Yaskawa INFORM job: X2_57-69(1)(90,0)_HARDOX.JBI

/JOB
//NAME X2_57-69(1)(90,0)_HARDOX
//POS
///NPOS 575,575,575,36,0,0
///TOOL 0
///POSTYPE PULSE
///PULSE
C00000=1941,-102693,-129564,10,101994,-18
C00001=-114160,-110711,-132276,13468,99543,32658
C00002=-115352,64839,21503,33302,71092,28193
C00003=-108531,78392,43986,16123,55140,37786
C00004=-108866,85252,55178,17040,51979,37122
C00005=-108996,88365,60166,17472,50599,36819
C00006=-108995,88536,62039,17737,49581,36632
C00007=-109034,88718,61766,17697,49840,36662
C00008=-109565,92254,66229,18307,49070,36272
C00009=-109034,88718,61766,17697,49840,36662
C00010=-108904,85509,56654,17244,51243,36976
C00011=-108571,78466,45235,16289,54445,37659
C00012=-107997,64928,29160,15382,57165,38310
C00013=-122208,49017,56535,29995,44799,-20500
C00014=-121054,58896,69591,30976,41821,-21001
C00015=-120607,61403,73283,31313,40811,-21157
C00016=-120607,63170,76793,32085,39739,-21613
C00017=-120607,62274,75028,31694,40274,-21383
C00018=-120608,64965,78215,32056,39778,-21596
C00019=-120607,62274,75028,31694,40274,-21383
C00020=-121364,56707,67057,30894,42308,-20982
C00021=-122534,47142,54464,30007,45185,-20534
C00022=-121995,48000,54847,25969,42983,-17450
C00023=-121016,58047,68030,26856,40021,-17900
C00024=-120639,62684,74202,27406,38635,-18182
C00025=-120639,64991,78769,28376,37190,-18734
C00026=-120639,62684,74202,27406,38635,-18182
C00027=-120856,61874,74409,27857,38220,-18464
C00028=-120445,66454,79858,28202,37199,-18614
C00029=-120856,61874,74409,27857,38220,-18464
C00030=-121238,57224,68232,27288,39602,-18174
C00031=-122229,47153,55046,26369,42553,-17714
C00032=-125892,1211,1187,22441,56600,-15676
C00033=-137814,-110158,-69296,24031,60757,-19595
C00034=-137728,-112604,-73316,23755,61850,-19313
C00035=-105364,-57557,-72999,2137,103390,46474
C00036=-115634,-1069,-31686,2185,107255,43060
C00037=-118085,-9413,-35378,2154,105305,42191
C00038=-118085,-9697,-34142,2144,104400,42176
C00039=-118085,-9660,-34317,2144,104526,42177
C00040=-119256,-9729,-34371,2141,104555,41779
C00041=-118897,-9712,-34357,2142,104546,41900
C00042=-118842,-14639,-38555,2142,104596,41919
C00043=-120602,-14747,-38323,2136,104444,41320
C00044=-120602,-13691,-37523,2136,104492,41320
C00045=-120602,-14272,-38765,2141,104957,41329
C00046=-118914,16972,-18491,2200,108489,41969
C00047=-117885,44382,12736,2123,103335,42227
C00048=-118751,44086,13966,2114,102449,41917
C00049=-118751,43916,15366,2106,101498,41903
C00050=-118751,43947,15080,2107,101690,41906
C00051=-119535,43897,15027,2105,101717,41640
C00052=-118660,44084,14052,2114,102390,41948
C00053=-117266,9455,-21352,2173,106346,42489
C00054=-117960,10005,-18871,2157,105121,42232
C00055=-117960,9788,-17905,2150,104416,42222
C00056=-117960,9832,-18111,2152,104564,42225
C00057=-119133,9750,-18184,2151,104599,41827
C00058=-118065,10242,-19838,2168,105841,42211
C00059=-118344,37722,-10535,2304,114239,18149
C00060=-118344,37722,-10535,2304,114239,-9791
C00061=-118344,37722,-10535,2304,91932,-69227
C00062=-118057,36728,-9901,-15898,90565,-72906
C00063=-124690,36878,-9748,-13863,89447,-74870
C00064=-125711,47870,427,-20022,100421,-78286
C00065=-126617,46625,2928,-19712,98166,-78212
C00066=-126617,46154,3748,-19667,97464,-78100
C00067=-126616,46214,3639,-19671,97560,-78116
C00068=-126105,44250,1538,-19774,97945,-78006
C00069=-130834,16270,-22947,-10503,81163,-76491
C00070=-130240,16776,-22499,-10733,81221,-76303
C00071=-130834,16571,-23478,-10493,81637,-76531
C00072=-131370,9383,-27977,-16260,78843,-76537
C00073=-131370,8975,-27154,-16296,78153,-76446
C00074=-131370,9027,-27263,-16291,78243,-76458
C00075=-131518,11566,-25004,-16235,78132,-76492
C00076=-131370,9027,-27263,-16291,78243,-76458
C00077=-132977,7860,-28293,-15633,77980,-76959
C00078=-131370,9307,-27828,-16266,78716,-76522
C00079=-122012,12842,-31502,-19803,84485,-74326
C00080=-122012,12842,-31502,-19803,84485,-74326
C00081=-119946,1839,-34459,-20715,81343,-73118
C00082=-119946,1422,-33631,-20749,80663,-73001
C00083=-119946,1471,-33732,-20744,80745,-73014
C00084=-120414,3746,-31827,-20569,80632,-73154
C00085=-119946,1471,-33731,-20744,80745,-73014
C00086=-130666,4901,-34214,-1657,83498,-73725
C00087=-129717,5880,-33367,-2009,83503,-73430
C00088=-120411,3435,-35647,-20479,82691,-73505
C00089=-123377,35712,-8759,-20752,103203,-78015
C00090=-123377,35712,-8759,-20752,103203,-78015
C00091=-123377,35151,-7898,-20672,102434,-77880
C00092=-123377,35217,-8004,-20682,102528,-77896
C00093=-123032,33253,-10001,-20749,102814,-77829
C00094=-123377,35217,-8004,-20682,102528,-77896
C00095=-124617,7277,-31513,-18537,87356,-75496
C00096=-125486,6411,-32266,-18262,87197,-75758
C00097=-124034,25111,-19103,-19892,98282,-77292
C00098=-138286,19736,-25230,-18597,101765,-82781
C00099=-139019,19392,-24177,-18406,100832,-82879
C00100=-139019,19048,-23693,-18372,100380,-82810
C00101=-139019,19115,-23789,-18378,100469,-82824
C00102=-138733,16890,-25865,-18440,100655,-82756
C00103=-139019,19115,-23789,-18378,100469,-82824
C00104=-148681,-9689,-46202,-1769,83169,-81630
C00105=-147538,-9148,-45777,-2193,83212,-81274
C00106=-148681,-9489,-46523,-1768,83469,-81634
C00107=-146164,-19217,-50920,-12366,76791,-81583
C00108=-146164,-19609,-50092,-12399,76095,-81512
C00109=-146164,-19552,-50218,-12394,76199,-81523
C00110=-146291,-17352,-48598,-12332,76313,-81579
C00111=-146227,-19942,-50503,-12369,76166,-81540
C00112=-147006,-20177,-50674,-12036,76040,-81783
C00113=-147897,-20398,-50837,-11655,75903,-82065
C00114=-147006,-19883,-51298,-12011,76564,-81835
C00115=-146427,-15690,-53542,-12122,80105,-82001
C00116=-146969,1425,-40243,-1367,79119,-79945
C00117=-144686,1127,-36373,-2406,76633,-79189
C00118=-144686,503,-35222,-2413,75606,-79175
C00119=-144686,641,-35492,-2413,75844,-79178
C00120=-144296,-3511,-38926,-2590,75836,-79052
C00121=-144296,-3690,-38579,-2592,75529,-79045
C00122=-144498,-2214,-37368,-2500,75537,-79111
C00123=-144701,-2831,-40035,-2396,76857,-79201
C00124=-153238,-15902,-45841,-12806,65800,-84378
C00125=-152617,-17217,-44336,-13318,64330,-83987
C00126=-152617,-17517,-43346,-13402,63584,-83898
C00127=-152617,-17437,-43619,-13378,63789,-83922
C00128=-152421,-22078,-47006,-13522,63527,-83819
C00129=-152421,-22202,-46551,-13563,63190,-83778
C00130=-152438,-20565,-45369,-13541,63298,-83797
C00131=-152580,-20987,-46826,-13385,63937,-83926
C00132=-154783,-40455,-61981,-12201,62944,-84616
C00133=-154783,-40864,-60420,-12327,61798,-84491
C00134=-154783,-41124,-59200,-12428,60934,-84393
C00135=-154783,-41063,-59504,-12403,61147,-84418
C00136=-152360,-40978,-59451,-13805,61537,-83550
C00137=-152360,-41066,-58995,-13847,61219,-83509
C00138=-153473,-40883,-58880,-13201,61064,-83911
C00139=-153098,-40967,-60326,-13315,61948,-83876
C00140=-169234,-16286,-61298,12968,85350,-87708
C00141=-176944,51771,6509,16270,80043,-90766
C00142=-175584,58970,15892,12405,82098,-90729
C00143=-175584,58471,16898,12427,81244,-90815
C00144=-175584,58538,16756,12423,81362,-90803
C00145=-175497,61195,19784,12406,80863,-90825
C00146=-175583,58538,16759,12438,81362,-90802
C00147=-168381,55909,13794,-5779,79883,-75223
C00148=-169176,56215,14138,-5481,79777,-75473
C00149=-168381,56447,12778,-5766,80781,-75265
C00150=-168717,73846,30007,3804,89205,-89178
C00151=-168717,73499,30710,3804,88596,-89198
C00152=-168717,73540,30620,3804,88675,-89193
C00153=-168793,71056,27634,3823,89235,-89202
C00154=-168717,73540,30620,3804,88675,-89193
C00155=-173050,67061,24969,13193,85810,-87576
C00156=-172324,66679,24524,12986,85777,-87344
C00157=-173050,67500,24071,13186,86568,-87495
C00158=-159020,60616,9002,-2431,101880,-86822
C00159=-158791,58641,10338,-2451,100051,-86715
C00160=-158791,57927,11282,-2444,99105,-86700
C00161=-158791,58001,11179,-2444,99208,-86703
C00162=-158877,55601,8473,-2433,99638,-86739
C00163=-158791,58001,11179,-2444,99208,-86703
C00164=-166389,29268,-13939,12099,84481,-87034
C00165=-165362,29139,-14065,11731,84356,-86720
C00166=-166389,29843,-14777,12087,85274,-86957
C00167=-168101,32508,-13251,8701,86943,-88153
C00168=-168101,31796,-12263,8703,85980,-88221
C00169=-168101,31909,-12426,8703,86137,-88210
C00170=-168113,34589,-9708,8710,85845,-88235
C00171=-167998,32289,-12043,8668,86088,-88180
C00172=-162647,21052,-20406,-2140,79162,-88550
C00173=-163390,21250,-20220,-1826,79131,-88783
C00174=-162647,21510,-21118,-2136,79834,-88562
C00175=-171713,88888,42294,-4924,102711,-49051
C00176=-183434,69304,21781,-4068,104650,-52979
C00177=-184172,69401,22560,-3999,104187,-53203
C00178=-184172,68923,23286,-3988,103496,-53177
C00179=-184172,68963,23221,-3991,103557,-53179
C00180=-183398,68489,22559,-4056,103756,-52932
C00181=-184172,68963,23221,-3991,103557,-53179
C00182=-173144,55424,11916,-25339,98078,-53030
C00183=-173306,53739,10045,-25337,98292,-53134
C00184=-184172,68963,23221,-3991,103557,-53179
C00185=-174683,52284,7590,-20558,90834,-51552
C00186=-174683,51681,8611,-20548,89951,-51401
C00187=-174683,51761,8468,-20549,90073,-51423
C00188=-175494,52416,9191,-20335,89781,-51643
C00189=-174683,51761,8468,-20549,90073,-51423
C00190=-174543,53466,10356,-20583,89839,-51336
C00191=-174438,56042,13238,-20604,89444,-51233
C00192=-174543,54156,9188,-20598,90847,-51507
C00193=-160426,19849,-34491,-24758,102852,-49155
C00194=-102402,-48698,-67991,2144,104784,47502
C00195=-177118,-86899,-49314,70294,69346,55717
C00196=-162665,-62437,-38431,68363,61957,60420
C00197=-158949,-60049,-34374,68890,58994,60353
C00198=-157479,-59004,-32692,69121,57826,60324
C00199=-157483,-57954,-30366,69642,57492,59876
C00200=-157504,-58291,-30998,69516,57587,59981
C00201=-155795,-59629,-31689,69630,56353,60099
C00202=-157504,-58291,-30998,69516,57587,59981
C00203=-157484,-58197,-30924,69514,57575,59985
C00204=-156523,-55844,-29677,69224,57103,60350
C00205=-157484,-58197,-30924,69514,57575,59985
C00206=-162670,-61686,-36716,68690,61698,60098
C00207=-161856,-67053,-41033,60813,38521,63477
C00208=-158996,-62210,-35558,60803,36300,63693
C00209=-157898,-60236,-33315,60834,35435,63760
C00210=-157901,-59173,-30986,61942,34994,63152
C00211=-156769,-58533,-30874,61190,34419,63655
C00212=-156166,-58108,-30651,60848,34087,63889
C00213=-156769,-58791,-31436,60917,34526,63803
C00214=-161883,-66170,-39058,61667,38156,62985
C00215=-175307,-91794,-54277,68294,45083,57713
C00216=-192656,-55134,-37587,64210,60039,59083
C00217=-162159,-23717,-10104,69718,77823,43469
C00218=-159534,-21701,-5637,70155,75421,43047
C00219=-158490,-20805,-3772,70360,74468,42873
C00220=-158493,-19842,-1317,70611,74104,42419
C00221=-158430,-19960,-1760,70561,74138,42521
C00222=-157077,-18912,-994,70615,73251,42719
C00223=-158430,-19960,-1760,70561,74138,42521
C00224=-162097,-22978,-8198,69866,77487,43129
C00225=-164656,-6441,2331,68796,80646,40119
C00226=-162354,-4355,7073,69146,78392,39620
C00227=-161441,-2725,10948,69469,77194,39063
C00228=-161443,-1987,12871,69626,76894,38710
C00229=-161439,-2551,11387,69503,77124,38984
C00230=-160415,-1923,12464,69637,76311,38965
C00231=-159548,-1589,12743,69678,75730,39076
C00232=-160719,-2768,10769,69490,76742,39193
C00233=-164702,-5497,5223,68969,80178,39553
C00234=-192656,-55134,-37587,64210,60039,59083
C00235=-125486,-104854,-75041,22917,86800,-65584
C00236=-126033,-92220,-87194,23391,99857,-63257
C00237=-126008,-87407,-69757,22927,92227,-64737
C00238=-122771,-89042,-67284,23124,89141,-64144
C00239=-121425,-89554,-66224,23215,87919,-63888
C00240=-121418,-87602,-63818,23218,87477,-63971
C00241=-121371,-87768,-64101,23220,87545,-63941
C00242=-119041,-87737,-64090,23370,86898,-63214
C00243=-121371,-87768,-64101,23220,87545,-63941
C00244=-119842,-88584,-64995,23320,87236,-63441
C00245=-119807,-91269,-65466,23334,86221,-63626
C00246=-119842,-88584,-64995,23320,87236,-63441
C00247=-121199,-88128,-66077,23230,88448,-63702
C00248=-124465,-86636,-68609,23034,91510,-64308
C00249=-142854,-85767,-72329,35934,81198,-48667
C00250=-140267,-86079,-63689,45810,58760,-32657
C00251=-135996,-80956,-60126,44498,56909,-31284
C00252=-134384,-78850,-58646,43955,56229,-30750
C00253=-134256,-77036,-56222,44175,55757,-30924
C00254=-134288,-77408,-56713,44133,55854,-30891
C00255=-132164,-77894,-56932,43544,54718,-30303
C00256=-134288,-77408,-56713,44133,55854,-30891
C00257=-88320,-91033,-56979,-46001,31828,15275
C00258=-89280,-88900,-56774,-44237,32046,14267
C00259=-88320,-91033,-56979,-46001,31828,15275
C00260=-85210,-101515,-62011,-50678,31900,18023
C00261=-89666,-105996,-71374,-46997,57370,39665
C00262=-112926,-92756,-65130,-39557,61499,44934
C00263=-117841,-88867,-61535,-38560,59130,43528
C00264=-119732,-87223,-60045,-38129,58240,42969
C00265=-119742,-85223,-57591,-38309,57852,43124
C00266=-119765,-85676,-58172,-38256,57941,43076
C00267=-121812,-86923,-58375,-37936,56635,42605
C00268=-119765,-85676,-58172,-38256,57941,43076
C00269=-121275,-85554,-58782,-37706,57631,42461
C00270=-122404,-83336,-58379,-37071,57860,41818
C00271=-121275,-85554,-58782,-37706,57631,42461
C00272=-114616,-91226,-63955,-39185,60786,44412
C00273=-114645,-97965,-79407,-37345,65578,42515
C00274=-116729,-83918,-76551,-18553,86191,61698
C00275=-117159,-89242,-76095,-11181,89587,70256
C00276=-119083,-90759,-73003,-11190,86687,69852
C00277=-119889,-89726,-70248,-11201,85432,69686
C00278=-119897,-88175,-68603,-11203,85218,69702
C00279=-119889,-89726,-70248,-11201,85432,69686
C00280=-119873,-91603,-70614,-11208,84708,69757
C00281=-119889,-89726,-70248,-11201,85432,69686
C00282=-107060,-93796,-69139,-19617,83326,67746
C00283=-109561,-94345,-69347,-19648,82582,66969
C00284=-107060,-93796,-69139,-19617,83326,67746
C00285=-120981,-91693,-72872,-11196,85873,69270
C00286=-118990,-90334,-76042,-11186,88750,69699
C00287=-119015,-93571,-89875,-11280,95471,69085
C00288=-121827,-98987,-110994,4235,90756,33976
C00289=-126467,-111869,-98615,30475,51467,-26148
C00290=-122938,-103029,-94111,27808,51796,-24337
C00291=-121643,-99583,-92275,26825,51945,-23680
C00292=-121634,-97826,-90039,26985,51518,-23798
C00293=-121643,-99583,-92275,26825,51945,-23680
C00294=-130783,-80407,-84869,35916,67887,-27578
C00295=-128717,-80853,-85070,35145,66956,-27002
C00296=-130783,-80407,-84869,35916,67887,-27578
C00297=-107674,-109601,-92730,7088,37825,-14001
C00298=-108083,-105924,-92018,7248,39302,-14088
C00299=-107674,-109601,-92730,7088,37825,-14001
C00300=-110011,-124661,-99237,10171,34381,-15732
C00301=-126906,-107253,-113226,22382,79753,-37979
C00302=-126893,-93432,-102362,29867,101882,-55415
C00303=-122864,-96655,-100816,29402,98217,-54829
C00304=-121215,-97700,-100096,29236,96792,-54563
C00305=-121210,-96197,-97952,29195,96310,-54685
C00306=-121215,-97700,-100096,29236,96792,-54563
C00307=-121163,-96448,-98340,29200,96390,-54646
C00308=-118846,-96389,-98319,29071,95614,-53959
C00309=-121163,-96448,-98340,29200,96390,-54646
C00310=-120263,-97948,-99498,29148,96030,-54394
C00311=-120240,-102374,-100607,29046,94623,-54741
C00312=-120263,-97948,-99498,29148,96030,-54394
C00313=-125973,-93962,-101877,29758,101067,-55277
C00314=-118596,-129181,-126473,-9366,77401,-2206
C00315=-114435,-108672,-97735,-33612,57488,30842
C00316=-118529,-101099,-93472,-31282,56999,29098
C00317=-120051,-98101,-91728,-30387,56847,28447
C00318=-120058,-96382,-89499,-30544,56421,28577
C00319=-120051,-98101,-91728,-30387,56847,28447
C00320=-120087,-96650,-89858,-30501,56482,28544
C00321=-122421,-96636,-89851,-29327,55655,27727
C00322=-120087,-96650,-89858,-30501,56482,28544
C00323=-120936,-97217,-90733,-29999,56393,28182
C00324=-120939,-93406,-89800,-29561,57600,27814
C00325=-120936,-97217,-90733,-29999,56393,28182
C00326=-115418,-107792,-96770,-33217,56982,30555
C00327=-105146,-130010,-122753,-24377,88875,54529
C00328=-114428,-145611,-119705,-15408,97435,71230
C00329=-117464,-150573,-117642,-15685,93169,70698
C00330=-118771,-152166,-116683,-15828,91559,70446
C00331=-118800,-148516,-114162,-15837,91865,70397
C00332=-118771,-152166,-116683,-15828,91559,70446
C00333=-89023,-160145,-112498,-25773,88935,79257
C00334=-92598,-162169,-112911,-26414,87133,78351
C00335=-89023,-160145,-112498,-25773,88935,79257
C00336=-143634,-123316,-108912,-7172,105756,63537
C00337=-144414,-127929,-109749,-7250,103844,63374
C00338=-143634,-123316,-108912,-7172,105756,63537
C00339=-142718,-121013,-109514,-7059,107379,63770
C00340=-140567,-114497,-110685,-6827,111603,64303
C00341=-106156,-132360,-130153,-17350,90664,54849
C00342=-113451,-107662,-104229,-36971,70393,33800
C00343=-118206,-101735,-100389,-35240,68968,32234
C00344=-120007,-99320,-98805,-34543,68461,31631
C00345=-120014,-97721,-96632,-34652,68030,31771
C00346=-120007,-99320,-98805,-34543,68461,31631
C00347=-120011,-97828,-96896,-34630,68120,31742
C00348=-122349,-97818,-96890,-33771,67193,31043
C00349=-120011,-97828,-96896,-34630,68120,31742
C00350=-121054,-97492,-97790,-34094,68307,31234
C00351=-121054,-93214,-96669,-33787,69569,30828
C00352=-121054,-97492,-97790,-34094,68307,31234
C00353=-114636,-105862,-103272,-36519,70163,33365
C00354=-114279,-101889,-100082,-25331,80876,44864
C00355=-118566,-99424,-96391,-24445,78685,43735
C00356=-120245,-97521,-93811,-24102,77637,43327
C00357=-120247,-96657,-92660,-24122,77395,43376
C00358=-120219,-96976,-93108,-24119,77505,43364
C00359=-122549,-96954,-93097,-23561,76842,42630
C00360=-120219,-96976,-93108,-24119,77505,43364
C00361=-114306,-100541,-98340,-25348,80523,44930
C00362=-120621,-97394,-101621,-24202,63073,45941
C00363=-120621,-97613,-99404,-24510,61722,46250
C00364=-126885,-95808,-100508,-15136,62705,44325
C00365=-124891,-100138,-106487,-19050,76932,40471
C00366=-124330,-97085,-92322,-20020,71587,41486
C00367=-120096,-97587,-96517,-20033,105608,38386
C00368=-120621,-97666,-97219,-19653,110159,37614
C00369=-120621,-97564,-100279,-19942,111985,37290
C00370=-114267,-119022,-117316,-18586,97333,41934
C00371=-120586,-140068,-100376,-59799,22791,77658
C00372=-120585,-131836,-89399,-65340,21573,80326
C00373=-120301,-131910,-88922,-66286,21610,80804
C00374=-120198,-131934,-88749,-66625,21626,80975
C00375=-119916,-129593,-85873,-68118,21579,81715
C00376=-118482,-138777,-95380,-52510,29730,72880
C00377=-120255,-147562,-109916,-33672,49046,60189
C00378=-120254,-140089,-100414,-34669,47370,60868
C00379=-115468,-148569,-111904,-12737,99323,53877
C00380=-120588,-148294,-110670,-9262,106248,51768
C00381=-120588,-160541,-124626,-9395,108516,51590
C00382=-136842,-121669,-124376,16041,91150,-8624
C00383=-120606,-113410,-86554,36159,18075,-56282
C00384=-120605,-110678,-81352,39700,16640,-57934
C00385=-120584,-111701,-82271,39578,16661,-57878
C00386=-120580,-111920,-82466,39553,16665,-57867
C00387=-120605,-109556,-79302,41216,16112,-58638
C00388=-124077,-125780,-98632,32708,39047,-51685
C00389=-120496,-124050,-111043,24637,69959,-42697
C00390=-120664,-121871,-104765,25113,67511,-43309
C00391=-121671,-124094,-110510,20986,97112,-39569
C00392=-120608,-124256,-111795,20648,99670,-38855
C00393=-120609,-125131,-115147,20777,101183,-38590
C00394=-120610,-125783,-123647,21277,105768,-37763
C00395=-120668,-128769,-125921,-5871,89606,-827
C00396=-107053,-95803,-77707,-38578,68772,44507
C00397=-120618,-86239,-59568,-37363,57829,42393
C00398=-120528,-85716,-59123,-36997,58097,42691
C00399=-120619,-91352,-71155,-22510,73817,56639
C00400=-119738,-88100,-63683,-22964,71349,57460
C00401=-119548,-88867,-66660,-18371,78749,62657
C00402=-120622,-86591,-69531,-13569,88626,68335
C00403=-120425,-89920,-79314,-13611,92853,67941
C00404=-120620,-95688,-83779,-13612,92610,67900
C00405=-120653,-118153,-99445,8937,69074,27704
C00406=-120618,-86290,-59555,39610,31833,-26802
C00407=-120617,-83679,-54099,41791,30283,-27941
C00408=-120617,-83181,-53105,42201,30015,-28153
C00409=-120617,-83020,-52785,42335,29929,-28222
C00410=-120619,-93115,-75724,25664,64689,-43944
C00411=-120826,-86244,-59129,27057,59793,-46292
C00412=-121400,-88637,-64040,23275,84750,-62478
C00413=-120618,-88758,-64988,22876,88456,-64391
C00414=-120618,-90407,-68808,22886,89847,-64125
C00415=-120645,-96149,-85177,23134,96436,-62865
C00416=-120704,-139648,-98792,22953,83536,-65363
C00417=-201677,-83839,-16745,82551,61455,23328
C00418=-193287,-71994,-23753,71338,80116,26125
C00419=-188716,-68676,-18939,72756,76807,26050
C00420=-186807,-37234,2063,68557,93943,25131
C00421=-186791,-37375,1977,68560,93924,25125
C00422=-188875,-55332,-8770,71294,85660,29887
C00423=-186990,-46090,-3659,67979,93495,33535
C00424=-187169,-52287,-8326,67185,92343,33510
C00425=-188906,-62105,-11935,69333,88967,33384
C00426=-188683,-64142,-13243,69128,88603,33879
C00427=-187867,-62779,-12578,68415,90081,34352
C00428=-188794,-66315,-17993,66765,90030,34259
C00429=-197371,-61565,-20436,64467,96999,34726
C00430=-180892,-45026,-152,77390,64230,28169
C00431=-201677,-83839,-16745,82551,61455,23328
C00432=-102465,-98091,-57376,11154,53691,1192
C00433=-117523,-2788,-9530,25488,75365,-1139
C00434=-125139,57134,55592,35785,69072,-6421
C00435=-125133,64451,72830,37508,63513,-8429
C00436=-123932,76756,90632,38887,59314,-9544
C00437=-123464,84249,101464,39928,56909,-10353
C00438=-122296,71715,85090,35181,54513,-6915
C00439=-122189,68599,81314,33173,52324,-4280
C00440=-122589,68250,80867,31901,50792,-2732
C00441=-122908,67120,79438,30365,49475,-1044
C00442=-123218,66439,78655,28729,48083,651
C00443=-123718,66653,78885,28024,47440,1365
C00444=-121882,59213,71115,24134,43656,7775
C00445=-110842,52453,67135,-14467,33841,33723
C00446=-111073,52381,67059,-14368,33810,33647
C00447=-110346,48653,61790,-14496,35224,33792
C00448=-108666,36587,42456,-14007,41045,33643
C00449=-114621,109196,43725,31616,85766,30078
C00450=-108492,104701,44017,11484,73458,41705
C00451=-108890,108743,52585,11893,70378,41274
C00452=-108566,112524,59213,11878,68242,41168
C00453=-105655,126679,78153,10634,63557,41739
C00454=-105456,124563,73948,10396,65010,41943
C00455=-114621,109196,43725,31616,85766,30078
C00456=-117523,-2788,-9530,25488,75365,-1139
C00457=-102465,-98091,-57376,11154,53691,1192
C00458=-194924,-89332,-18186,86283,57168,22588
C00459=-189291,-99620,-43569,70052,49879,58298
C00460=-183385,-95654,-38841,71457,45923,58650
C00461=-179289,-94967,-37057,72626,43143,58783
C00462=-180541,-94166,-36956,72139,44032,58817
C00463=-181760,-88303,-31492,78702,40431,52425
C00464=-191947,-67176,-20621,75434,55592,47212
C00465=-188895,-71260,-14971,91913,47690,32624
C00466=-190378,-73018,-17241,90953,48654,32921
C00467=-194954,-78245,-22550,88961,51649,33203
C00468=-209629,-115340,-51402,66324,56026,36469
C00469=-117179,-93991,-70029,-10923,64438,-31948
C00470=-91116,-86743,-69135,-16598,71993,-23160
C00471=-103770,-45855,-47036,-2494,89723,45807
C00472=-108273,11270,-37038,-2487,112775,43845
C00473=-108273,11270,-37038,-2487,89909,-74519
C00474=-105376,-26657,-54571,-20367,72508,-76542
C00475=-105949,-25432,-50040,-20418,71411,-76593
C00476=-111295,-34234,-56012,-18069,69407,-78179
C00477=-111295,-34234,-56012,-18069,69407,-78179
C00478=-111814,5193,-34860,-16843,99127,-82784
C00479=-126499,17841,-26152,8088,107235,-84265
C00480=-125779,18021,-24749,13991,103199,-83193
C00481=-125779,18021,-24749,13991,103199,-83193
C00482=-129206,-19638,-47941,20123,76796,-86688
C00483=-105949,-25432,-50040,-20418,71411,-76593
C00484=-105772,-26518,-53791,-20314,73095,-76824
C00485=-110449,42794,4075,-18195,72061,-78293
C00486=-134580,44443,5827,-6280,68369,-86206
C00487=-132902,40830,5501,-11723,65791,-86256
C00488=-133811,44041,12444,-11477,63095,-86312
C00489=-132439,65612,31839,-21122,77005,-90132
C00490=-132439,65612,31839,-21122,77005,-90132
C00491=-131095,89890,59104,-25378,85140,-84106
C00492=-135491,96161,62942,-14320,88749,-84613
C00493=-136289,102154,69415,-9018,88918,-84466
C00494=-136256,109661,65993,-5037,95739,-84423
C00495=-136256,109661,65993,-5037,95739,-84423
C00496=-140207,76037,26999,-284,85486,-84853
C00497=-133811,44041,12444,-11477,63095,-86312
C00498=-133933,42277,8522,-11269,64556,-86504
C00499=-130781,23057,-17066,-12462,70742,-86033
C00500=-135329,-34726,-64223,-12702,72089,86721
C00501=-145906,18547,-31269,-17564,106398,77717
C00502=-147099,16763,-29681,-17191,104364,77630
C00503=-148291,15260,-26923,-15200,103832,76849
C00504=-153964,13497,-28672,-13715,103084,74443
C00505=-153964,13497,-28672,-13715,103084,74443
C00506=-157532,-15464,-48977,-8940,83674,75571
C00507=-162114,-25324,-53698,-902,74788,75797
C00508=-161555,-24902,-53581,2493,75208,76448
C00509=-171418,-6750,-41347,13698,82414,75012
C00510=-171418,-6750,-41347,13698,82414,75012
C00511=-169992,8963,-31883,12281,94308,76305
C00512=-148291,15260,-26923,-15200,103832,76849
C00513=-148064,18239,-27550,-15385,105723,76679
C00514=-181534,55879,5002,-6914,99225,-52479
C00515=-183067,52708,5629,-4970,98839,-52617
C00516=-181530,67422,22384,-5485,96546,-51647
C00517=-181530,67422,22384,-5485,96546,-51647
C00518=-175010,45086,3284,-19371,84208,-50498
C00519=-167011,75857,41236,-38328,94510,-53164
C00520=-166996,74549,39713,-38471,94870,-53286
C00521=-166862,63292,26956,-39810,97835,-54325
C00522=-166862,63293,26956,-39810,97835,-54325
C00523=-174268,85207,46337,-23890,107283,-57472
C00524=-183067,52708,5629,-4970,98839,-52617
C00525=-182882,56404,7954,-5014,99317,-52578
C00526=-165691,102270,54007,-6025,95854,-77116
C00527=-174763,100788,53636,151,98660,-79371
C00528=-175780,100346,53981,269,98225,-79701
C00529=-172514,98622,51828,866,99394,-78489
C00530=-172514,98622,51828,866,99394,-78489
C00531=-178493,70544,26694,14946,87921,-78994
C00532=-175677,45540,12642,8743,69973,-81130
C00533=-173166,43222,10537,1232,68328,-81339
C00534=-173957,38496,8010,-2752,63398,-82249
C00535=-173957,38496,8010,-2752,63398,-82249
C00536=-168220,64807,30846,-15967,78983,-83071
C00537=-175780,100346,53981,269,98225,-79701
C00538=-174777,101613,54080,153,98812,-79373
C00539=-163509,93679,42010,-1155,102230,-75733
C00540=-166182,93539,45341,1617,101458,-76190
C00541=-163160,91310,42596,3283,101462,-74900
C00542=-163160,91310,42596,3283,101462,-74900
C00543=-169452,54644,10871,16856,84100,-76164
C00544=-159291,36753,-4751,-4537,72622,-76986
C00545=-157932,36959,-4072,-9427,72445,-77153
C00546=-160362,40124,-1567,-9930,74025,-78463
C00547=-160362,40124,-1567,-9930,74025,-78463
C00548=-160290,65148,19778,-11331,88559,-79894
C00549=-166167,93639,45471,1615,101430,-76186
C00550=-166035,95428,45416,1610,102379,-76130
C00551=-166063,-1948,-41107,-10479,80074,-77808
C00552=-166651,-13744,-43383,-12910,70088,-77581
C00553=-166009,6948,-26476,-13209,70411,-77394
C00554=-166009,6948,-26476,-13209,70411,-77394
C00555=-169595,16125,-21731,-5794,76487,-77956
C00556=-176822,20131,-18643,8586,78706,-78235
C00557=-160365,16055,-22103,5880,77875,-72175
C00558=-161224,13274,-26949,6213,79478,-72370
C00559=-143929,-35419,-63325,-1105,76336,-66923
C00560=-118137,-166394,-107438,-18333,39307,-53291
C00561=-136403,-175311,-100414,52501,46046,31610
C00562=-136403,-175311,-100414,52501,46046,31610
C00563=-146221,-138467,-86930,47519,55366,36499
C00564=-143930,-139137,-87070,47419,54034,37009
C00565=-143930,-139137,-87070,47419,54034,37009
C00566=-170274,-134580,-90328,36528,58155,28961
C00567=-133594,-133818,-95395,2291,53248,46023
C00568=-127891,-62902,-68366,-13,72975,48365
C00569=-125715,-6143,-31037,-736,79177,49082
C00570=-125715,-6143,-31037,-736,79177,49082
C00571=-121975,46893,6489,-8294,110832,47946
C00572=-123069,51099,10752,-9131,109699,67175
C00573=-123053,53405,11005,-9199,110717,67100
C00574=-126089,-90466,-96021,-8826,102422,66678
BC00000=210618,668760,578653
BC00001=307087,668760,191900
BC00002=307087,789553,191900
BC00003=307087,789553,191900
BC00004=307087,789553,191900
BC00005=307087,789553,191900
BC00006=307087,789553,191900
BC00007=307087,789553,191900
BC00008=307087,789553,191900
BC00009=307087,789553,191900
BC00010=307087,789553,191900
BC00011=307087,789553,191900
BC00012=307087,789553,191900
BC00013=319173,776954,280603
BC00014=319173,776954,280603
BC00015=319173,776954,280603
BC00016=319173,776954,280603
BC00017=319173,776954,280603
BC00018=319173,776954,280603
BC00019=319173,776954,280603
BC00020=319173,776954,280603
BC00021=319173,776954,280603
BC00022=324465,771616,271785
BC00023=324465,771616,271785
BC00024=324465,771616,271785
BC00025=324465,771616,271785
BC00026=324465,771616,271785
BC00027=324465,771616,271785
BC00028=324465,771616,271785
BC00029=324465,771616,271785
BC00030=324465,771616,271785
BC00031=324465,771616,271785
BC00032=324465,747237,368530
BC00033=324465,670069,674761
BC00034=169071,670069,459913
BC00035=137209,684775,182974
BC00036=137209,684775,182974
BC00037=137209,684775,182974
BC00038=137209,684775,182974
BC00039=137209,684775,182974
BC00040=137209,684775,182974
BC00041=137209,684775,182974
BC00042=137209,684775,182974
BC00043=137209,684775,182974
BC00044=137209,684775,182974
BC00045=137209,684775,182974
BC00046=137209,684775,182974
BC00047=137210,684774,182973
BC00048=137210,684774,182973
BC00049=137210,684774,182973
BC00050=137210,684774,182973
BC00051=137210,684774,182973
BC00052=137210,684774,182973
BC00053=136881,774000,182759
BC00054=136881,774000,182759
BC00055=136881,774000,182759
BC00056=136881,774000,182759
BC00057=136881,774000,182759
BC00058=136881,774000,182759
BC00059=136881,774000,73910
BC00060=136881,774000,73910
BC00061=136881,774000,73910
BC00062=136881,774000,73910
BC00063=156999,774000,73910
BC00064=156999,774000,73910
BC00065=156999,774000,73910
BC00066=156999,774000,73910
BC00067=156998,774000,73899
BC00068=156998,774000,73898
BC00069=156998,774000,73899
BC00070=156998,774000,73899
BC00071=156998,774000,73899
BC00072=156998,774000,73898
BC00073=156998,774000,73898
BC00074=156998,774000,73898
BC00075=156998,774000,73898
BC00076=156998,774000,73898
BC00077=156998,774000,73898
BC00078=156998,774000,73898
BC00079=156998,774000,73898
BC00080=156998,712221,73898
BC00081=156998,712221,73898
BC00082=156998,712221,73898
BC00083=156998,712221,73898
BC00084=156998,712221,73898
BC00085=156998,712221,73898
BC00086=156998,712221,73898
BC00087=156998,712221,73898
BC00088=156998,712221,73898
BC00089=156998,712221,73898
BC00090=156998,712221,73898
BC00091=156998,712221,73898
BC00092=156998,712221,73898
BC00093=156998,712221,73898
BC00094=156998,712221,73898
BC00095=156998,712221,73898
BC00096=156998,712221,73898
BC00097=156998,712221,73898
BC00098=156998,712221,73898
BC00099=156998,712221,73898
BC00100=156998,712221,73898
BC00101=156998,712221,73898
BC00102=156998,712221,73898
BC00103=156998,712221,73898
BC00104=156998,712221,73898
BC00105=156998,712221,73898
BC00106=156998,712221,73898
BC00107=156998,712221,73898
BC00108=156998,712221,73898
BC00109=156998,712221,73898
BC00110=156998,712221,73898
BC00111=156998,712221,73898
BC00112=156998,712221,73898
BC00113=156998,712221,73898
BC00114=156998,712221,73898
BC00115=156998,747592,73898
BC00116=156998,747592,73897
BC00117=156998,747592,73897
BC00118=156998,747592,73897
BC00119=156998,747592,73897
BC00120=156998,747592,73897
BC00121=156998,747592,73897
BC00122=156998,747592,73897
BC00123=156998,747592,73897
BC00124=156998,747592,73897
BC00125=156998,747592,73897
BC00126=156998,747592,73897
BC00127=156998,747592,73897
BC00128=156998,747592,73897
BC00129=156998,747592,73897
BC00130=156998,747592,73897
BC00131=156998,747592,73897
BC00132=156998,747592,73897
BC00133=156998,747592,73897
BC00134=156998,747592,73897
BC00135=156998,747592,73897
BC00136=156998,747592,73897
BC00137=156998,747592,73897
BC00138=156998,747592,73897
BC00139=156998,747592,73897
BC00140=156998,781832,73897
BC00141=186269,781832,57715
BC00142=186269,781832,55591
BC00143=186269,781832,55591
BC00144=186269,781832,55591
BC00145=186269,781832,55591
BC00146=186269,781832,55589
BC00147=186269,781832,55589
BC00148=186269,781832,55589
BC00149=186269,781832,55589
BC00150=186269,781832,55591
BC00151=186269,781832,55591
BC00152=186269,781832,55591
BC00153=186269,781832,55591
BC00154=186269,781832,55591
BC00155=186269,781832,55591
BC00156=186269,781832,55591
BC00157=186269,781832,55591
BC00158=186269,766875,55591
BC00159=186269,766875,55591
BC00160=186269,766875,55591
BC00161=186269,766875,55591
BC00162=186269,766875,55591
BC00163=186269,766875,55591
BC00164=186269,766875,55591
BC00165=186269,766875,55591
BC00166=186269,766875,55591
BC00167=186269,766875,55591
BC00168=186269,766875,55591
BC00169=186269,766875,55591
BC00170=186269,766875,55591
BC00171=186269,766875,55591
BC00172=186269,766875,55591
BC00173=186269,766875,55591
BC00174=186269,766875,55591
BC00175=221494,747543,55591
BC00176=221494,747543,55591
BC00177=221494,747543,55591
BC00178=221494,747543,55591
BC00179=221494,747543,55591
BC00180=221494,747543,55591
BC00181=221494,747543,55591
BC00182=221494,747543,55591
BC00183=221494,747543,55591
BC00184=221494,747543,55591
BC00185=221494,747543,55591
BC00186=221494,747543,55591
BC00187=221494,747543,55591
BC00188=221494,747543,55591
BC00189=221494,747543,55591
BC00190=221494,747543,55591
BC00191=221494,747543,55590
BC00192=221494,747543,55591
BC00193=221494,747543,55591
BC00194=136881,673536,182759
BC00195=33003,666220,204314
BC00196=33003,666220,204314
BC00197=33003,666220,204314
BC00198=33003,666220,204314
BC00199=33003,666220,204314
BC00200=33003,666220,204314
BC00201=33003,666220,204314
BC00202=33003,666220,204314
BC00203=33003,666220,204314
BC00204=33003,666220,204314
BC00205=33003,666220,204314
BC00206=33003,666220,204314
BC00207=48470,666220,217137
BC00208=48470,666220,217137
BC00209=48470,666220,217137
BC00210=48470,666220,217137
BC00211=48470,666220,217137
BC00212=48470,666220,217137
BC00213=48470,666220,217137
BC00214=48470,666220,217137
BC00215=48470,666220,217137
BC00216=48470,666220,217137
BC00217=15,666220,230034
BC00218=15,666220,230034
BC00219=15,666220,230034
BC00220=15,666220,230034
BC00221=15,666220,230034
BC00222=15,666220,230034
BC00223=15,666220,230034
BC00224=15,666220,230034
BC00225=15,666220,235835
BC00226=15,666220,235835
BC00227=15,666220,235835
BC00228=15,666220,235835
BC00229=15,666220,235835
BC00230=15,666221,235834
BC00231=15,666220,235835
BC00232=15,666220,235835
BC00233=15,666220,235835
BC00234=48470,666220,217137
BC00235=32831,670161,1075175
BC00236=32831,729596,1075175
BC00237=32831,729596,1075175
BC00238=32831,729596,1075175
BC00239=32831,729596,1075175
BC00240=32831,729596,1075175
BC00241=32831,729596,1075175
BC00242=32831,729596,1075175
BC00243=32831,729596,1075175
BC00244=32831,729596,1075175
BC00245=32831,729596,1075175
BC00246=32831,729596,1075175
BC00247=32831,729596,1075175
BC00248=32831,729596,1075175
BC00249=37728,721693,1075175
BC00250=41810,715107,1075175
BC00251=41810,715107,1075175
BC00252=41810,715107,1075175
BC00253=41810,715107,1075175
BC00254=41810,715107,1075175
BC00255=41810,715107,1075175
BC00256=41810,715107,1075175
BC00257=41810,715107,1075175
BC00258=41810,715107,1075175
BC00259=41810,715107,1075175
BC00260=41810,715107,1075175
BC00261=53876,706752,1075175
BC00262=60427,702216,1075175
BC00263=60427,702216,1075175
BC00264=60427,702216,1075175
BC00265=60427,702216,1075175
BC00266=60427,702216,1075175
BC00267=60427,702216,1075175
BC00268=60427,702216,1075175
BC00269=60427,702216,1075175
BC00270=60427,702216,1075175
BC00271=60427,702216,1075175
BC00272=60427,702216,1075175
BC00273=60427,702216,1075175
BC00274=46834,716034,1075175
BC00275=41397,721561,1075175
BC00276=41397,721561,1075175
BC00277=41397,721561,1075175
BC00278=41397,721561,1075175
BC00279=41397,721561,1075175
BC00280=41397,721561,1075175
BC00281=41397,721561,1075175
BC00282=41397,721561,1075175
BC00283=41397,721561,1075175
BC00284=41397,721561,1075175
BC00285=41397,721561,1075175
BC00286=41397,721561,1075175
BC00287=41397,721561,1075175
BC00288=77086,766277,1075175
BC00289=137161,841550,1075175
BC00290=137161,841550,1075175
BC00291=137161,841550,1075175
BC00292=137161,841550,1075175
BC00293=137161,841550,1075175
BC00294=137161,841550,1075175
BC00295=137161,841550,1075175
BC00296=137161,841550,1075175
BC00297=137161,841550,1075175
BC00298=137161,841550,1075175
BC00299=137161,841550,1075175
BC00300=137161,841550,1075175
BC00301=128673,864447,1075175
BC00302=121183,884651,1075175
BC00303=121183,884651,1075175
BC00304=121183,884651,1075175
BC00305=121183,884651,1075175
BC00306=121183,884651,1075175
BC00307=121183,884651,1075175
BC00308=121183,884651,1075175
BC00309=121183,884651,1075175
BC00310=121183,884651,1075175
BC00311=121183,884651,1075175
BC00312=121183,884651,1075175
BC00313=121183,884651,1075175
BC00314=162519,857645,1075175
BC00315=188050,840965,1075175
BC00316=188050,840965,1075175
BC00317=188050,840965,1075175
BC00318=188050,840965,1075175
BC00319=188050,840965,1075175
BC00320=188050,840965,1075175
BC00321=188050,840965,1075175
BC00322=188050,840965,1075175
BC00323=188050,840965,1075175
BC00324=188050,840965,1075175
BC00325=188050,840965,1075175
BC00326=188050,840965,1075175
BC00327=177981,881480,1075175
BC00328=169709,914761,1075175
BC00329=169709,914761,1075175
BC00330=169709,914761,1075175
BC00331=169709,914761,1075175
BC00332=169709,914761,1075175
BC00333=169709,914761,1075175
BC00334=169709,914761,1075175
BC00335=169709,914761,1075175
BC00336=169709,914761,1075175
BC00337=169709,914761,1075175
BC00338=169709,914761,1075175
BC00339=169709,914761,1075175
BC00340=169709,914761,1075175
BC00341=159152,880596,1075175
BC00342=150354,852125,1075175
BC00343=150354,852125,1075175
BC00344=150354,852125,1075175
BC00345=150354,852125,1075175
BC00346=150354,852125,1075175
BC00347=150354,852125,1075175
BC00348=150354,852125,1075175
BC00349=150354,852125,1075175
BC00350=150354,852125,1075175
BC00351=150354,852125,1075175
BC00352=150354,852125,1075175
BC00353=150354,852125,1075175
BC00354=138535,800539,1075175
BC00355=138535,800539,1075175
BC00356=138535,800539,1075175
BC00357=138535,800539,1075175
BC00358=138535,800539,1075175
BC00359=138535,800539,1075175
BC00360=138535,800539,1075175
BC00361=138535,800539,1075175
BC00362=139926,838224,1075175
BC00363=134477,841860,1075175
BC00364=132297,843314,1075175
BC00365=135301,861824,1075175
BC00366=135628,791701,1075175
BC00367=127557,845014,1075175
BC00368=128457,853081,1075175
BC00369=133547,854476,1075175
BC00370=133547,854476,1075175
BC00371=185526,847143,1075175
BC00372=185547,847145,1075175
BC00373=180367,852195,1075175
BC00374=178499,854016,1075175
BC00375=178499,854016,1075175
BC00376=181436,863252,1075175
BC00377=187425,882089,1075175
BC00378=187544,843803,1075173
BC00379=163075,924936,1075175
BC00380=160150,941259,1075175
BC00381=163894,945401,1075175
BC00382=155016,866117,1075175
BC00383=147551,828920,1075175
BC00384=147562,828921,1075175
BC00385=152516,835936,1075175
BC00386=153570,837428,1075175
BC00387=153570,837428,1075175
BC00388=143866,860842,1075175
BC00389=131316,891124,1075175
BC00390=131456,861099,1075175
BC00391=136555,907393,1075175
BC00392=134846,911418,1075175
BC00393=129544,912127,1075175
BC00394=129523,912125,1075175
BC00395=99118,813312,1075175
BC00396=64307,700180,1075175
BC00397=58098,703250,1075175
BC00398=55325,704971,1075175
BC00399=41598,728447,1075175
BC00400=60495,698876,1075175
BC00401=53827,709917,1075175
BC00402=47010,724325,1075175
BC00403=50143,727052,1075175
BC00404=50122,727050,1075175
BC00405=43900,716168,1075175
BC00406=35524,701519,1075175
BC00407=35534,701520,1075175
BC00408=39202,708199,1075175
BC00409=40669,710870,1075175
BC00410=31604,749687,1075172
BC00411=32090,681060,1075175
BC00412=35435,723771,1075175
BC00413=34090,730815,1075175
BC00414=29574,733664,1075175
BC00415=29574,733664,1075175
BC00416=29574,668853,1075175
BC00417=15,675786,401985
BC00418=15,747285,294679
BC00419=15,747285,294679
BC00420=15,747285,294679
BC00421=15,747285,294679
BC00422=15,747285,294679
BC00423=15,747285,294679
BC00424=15,747285,294679
BC00425=15,747285,294679
BC00426=15,747285,294679
BC00427=15,747285,294679
BC00428=15,747285,294679
BC00429=15,747285,294679
BC00430=15,675786,401985
BC00431=15,675786,401985
BC00432=281438,669247,530529
BC00433=311998,746592,376004
BC00434=327524,785889,297495
BC00435=327524,785889,297495
BC00436=327524,785889,297495
BC00437=327524,785889,297495
BC00438=327524,785889,297495
BC00439=327524,785889,297495
BC00440=327524,785889,297495
BC00441=327524,785889,297495
BC00442=327524,785889,297495
BC00443=327524,785889,297495
BC00444=327524,785889,297495
BC00445=327524,785889,297495
BC00446=327524,785889,297495
BC00447=327524,785889,297495
BC00448=327524,785889,297495
BC00449=301537,784116,209
BC00450=301537,784116,209
BC00451=301537,784116,209
BC00452=301537,784116,209
BC00453=301537,784116,209
BC00454=301537,784116,209
BC00455=301537,784116,209
BC00456=311998,746592,376004
BC00457=281438,669247,530529
BC00458=28742,675786,401985
BC00459=69504,715923,290542
BC00460=69504,715923,290542
BC00461=69504,715923,290542
BC00462=69504,715923,290542
BC00463=69504,715923,290542
BC00464=69504,715923,290542
BC00465=69504,715923,290542
BC00466=69504,715923,290542
BC00467=69504,715923,290542
BC00468=69504,715923,290542
BC00469=108267,707570,269586
BC00470=108267,707570,269586
BC00471=115634,729988,290459
BC00472=115634,729988,82791
BC00473=115634,729988,82791
BC00474=115634,729988,82791
BC00475=115634,729988,82791
BC00476=115634,729988,82791
BC00477=115634,729988,82791
BC00478=115634,729988,82791
BC00479=115634,729988,82791
BC00480=115634,729988,82791
BC00481=115634,729988,82791
BC00482=115634,729988,82791
BC00483=115634,729988,82791
BC00484=115634,729988,82791
BC00485=115634,729988,82791
BC00486=177007,729988,82791
BC00487=177007,729988,82791
BC00488=177007,729988,82791
BC00489=176923,729988,82791
BC00490=176923,729988,82791
BC00491=176923,729988,82791
BC00492=176923,729988,82791
BC00493=176882,729988,82791
BC00494=176882,729988,787
BC00495=176882,729988,787
BC00496=186092,729988,787
BC00497=177007,729988,82791
BC00498=177007,729988,82791
BC00499=177007,729988,82791
BC00500=177007,729988,82791
BC00501=177007,729988,82791
BC00502=177007,729988,82791
BC00503=176711,729988,82791
BC00504=176429,729988,82791
BC00505=176429,729988,82791
BC00506=176429,729988,82791
BC00507=176429,729988,82791
BC00508=176365,729988,82791
BC00509=194916,729988,82791
BC00510=194916,729988,82791
BC00511=194916,729988,82791
BC00512=176711,729988,82791
BC00513=176711,729988,82791
BC00514=221494,747543,55589
BC00515=221494,747543,55588
BC00516=221330,747479,55687
BC00517=221330,747479,55687
BC00518=221330,747479,55687
BC00519=221330,747479,55687
BC00520=221325,747477,55690
BC00521=221284,747461,55715
BC00522=221284,747461,55715
BC00523=221284,747461,55715
BC00524=221494,747543,55588
BC00525=221494,747543,55588
BC00526=200576,765754,2878
BC00527=201503,792313,2878
BC00528=201503,792313,2878
BC00529=201503,792313,2878
BC00530=201503,792313,2878
BC00531=201013,792117,38546
BC00532=201503,792313,100685
BC00533=201503,792313,100685
BC00534=201503,792313,100685
BC00535=201503,792313,100685
BC00536=201503,792313,100685
BC00537=201503,792313,2878
BC00538=201503,792313,2878
BC00539=201213,748947,2878
BC00540=201213,748947,2878
BC00541=201213,748947,2878
BC00542=201213,748947,2878
BC00543=202078,748947,38400
BC00544=202078,748947,38400
BC00545=202039,748918,38467
BC00546=202039,748918,38467
BC00547=202039,748918,38467
BC00548=202039,748918,38467
BC00549=201213,748947,2878
BC00550=201213,748947,2878
BC00551=201213,748947,74226
BC00552=201214,748947,74225
BC00553=201214,748947,74225
BC00554=201214,748947,74225
BC00555=201214,748947,74225
BC00556=201214,748947,74225
BC00557=201214,748947,74225
BC00558=201214,748947,74225
BC00559=170128,748947,109531
BC00560=170128,748947,149986
BC00561=108120,704448,149986
BC00562=108120,748947,149986
BC00563=106324,748947,149986
BC00564=106324,748947,149986
BC00565=106324,748947,149986
BC00566=161663,748947,149986
BC00567=161663,748947,149986
BC00568=161663,748947,149986
BC00569=161663,748947,149986
BC00570=161663,748947,149986
BC00571=161663,748947,96847
BC00572=161663,748947,96847
BC00573=161663,748947,96847
BC00574=161663,692365,96847
EC00000=798156,0
EC00001=798156,0
EC00002=798156,0
EC00003=798156,0
EC00004=798156,0
EC00005=798156,0
EC00006=798156,0
EC00007=798156,0
EC00008=798156,0
EC00009=798156,0
EC00010=798156,0
EC00011=798156,0
EC00012=798156,0
EC00013=798156,0
EC00014=798156,0
EC00015=798156,0
EC00016=798156,0
EC00017=798156,0
EC00018=798156,0
EC00019=798156,0
EC00020=798156,0
EC00021=798156,0
EC00022=798156,0
EC00023=798156,0
EC00024=798156,0
EC00025=798156,0
EC00026=798156,0
EC00027=798156,0
EC00028=798156,0
EC00029=798156,0
EC00030=798156,0
EC00031=798156,0
EC00032=798156,0
EC00033=798156,0
EC00034=798156,0
EC00035=798156,0
EC00036=798156,0
EC00037=798156,0
EC00038=798156,0
EC00039=798156,0
EC00040=798156,0
EC00041=798156,0
EC00042=798156,0
EC00043=798156,0
EC00044=798156,0
EC00045=798156,0
EC00046=798156,0
EC00047=798155,1
EC00048=798155,1
EC00049=798155,1
EC00050=798155,1
EC00051=798155,1
EC00052=798155,1
EC00053=798156,0
EC00054=798156,0
EC00055=798156,0
EC00056=798156,0
EC00057=798156,0
EC00058=798156,0
EC00059=798156,0
EC00060=798156,0
EC00061=798156,0
EC00062=798156,0
EC00063=798156,0
EC00064=798156,0
EC00065=798156,0
EC00066=798156,0
EC00067=798154,1
EC00068=798153,2
EC00069=798154,1
EC00070=798154,1
EC00071=798154,1
EC00072=798153,2
EC00073=798153,2
EC00074=798153,2
EC00075=798153,2
EC00076=798153,2
EC00077=798153,2
EC00078=798153,2
EC00079=798153,2
EC00080=798153,2
EC00081=798153,2
EC00082=798153,2
EC00083=798153,2
EC00084=798153,2
EC00085=798153,2
EC00086=798153,2
EC00087=798153,2
EC00088=798153,2
EC00089=798153,2
EC00090=798153,2
EC00091=798153,2
EC00092=798153,2
EC00093=798153,2
EC00094=798153,2
EC00095=798153,2
EC00096=798153,2
EC00097=798153,2
EC00098=798153,2
EC00099=798153,2
EC00100=798153,2
EC00101=798153,2
EC00102=798153,2
EC00103=798153,2
EC00104=798153,2
EC00105=798153,2
EC00106=798153,2
EC00107=798153,2
EC00108=798153,2
EC00109=798153,2
EC00110=798153,2
EC00111=798153,2
EC00112=798153,2
EC00113=798153,2
EC00114=798153,2
EC00115=798153,2
EC00116=798153,3
EC00117=798153,3
EC00118=798153,3
EC00119=798153,3
EC00120=798153,3
EC00121=798153,3
EC00122=798153,3
EC00123=798153,3
EC00124=798153,3
EC00125=798153,3
EC00126=798153,3
EC00127=798153,3
EC00128=798153,3
EC00129=798153,3
EC00130=798153,3
EC00131=798153,3
EC00132=798153,3
EC00133=798153,3
EC00134=798153,3
EC00135=798153,3
EC00136=798153,3
EC00137=798153,3
EC00138=798153,3
EC00139=798153,3
EC00140=798153,3
EC00141=798153,3
EC00142=798151,4
EC00143=798151,4
EC00144=798151,4
EC00145=798151,4
EC00146=798151,4
EC00147=798151,4
EC00148=798151,4
EC00149=798151,4
EC00150=798151,4
EC00151=798151,4
EC00152=798151,4
EC00153=798151,4
EC00154=798151,4
EC00155=798151,4
EC00156=798151,4
EC00157=798151,4
EC00158=798151,4
EC00159=798151,4
EC00160=798151,4
EC00161=798151,4
EC00162=798151,4
EC00163=798151,4
EC00164=798151,4
EC00165=798151,4
EC00166=798151,4
EC00167=798151,4
EC00168=798151,4
EC00169=798151,4
EC00170=798151,4
EC00171=798151,4
EC00172=798151,4
EC00173=798151,4
EC00174=798151,4
EC00175=798151,4
EC00176=798151,4
EC00177=798151,4
EC00178=798151,4
EC00179=798151,4
EC00180=798151,4
EC00181=798151,4
EC00182=798151,4
EC00183=798151,4
EC00184=798151,4
EC00185=798151,4
EC00186=798151,4
EC00187=798151,4
EC00188=798151,4
EC00189=798151,4
EC00190=798151,4
EC00191=798150,5
EC00192=798151,4
EC00193=798151,4
EC00194=798156,0
EC00195=798156,0
EC00196=798156,0
EC00197=798156,0
EC00198=798156,0
EC00199=798156,0
EC00200=798156,0
EC00201=798156,0
EC00202=798156,0
EC00203=798156,0
EC00204=798156,0
EC00205=798156,0
EC00206=798156,0
EC00207=798156,0
EC00208=798156,0
EC00209=798156,0
EC00210=798156,0
EC00211=798156,0
EC00212=798156,0
EC00213=798156,0
EC00214=798156,0
EC00215=798156,0
EC00216=798156,0
EC00217=798156,0
EC00218=798156,0
EC00219=798156,0
EC00220=798156,0
EC00221=798156,0
EC00222=798156,0
EC00223=798156,0
EC00224=798156,0
EC00225=798156,0
EC00226=798156,0
EC00227=798156,0
EC00228=798156,0
EC00229=798156,0
EC00230=798155,0
EC00231=798156,0
EC00232=798156,0
EC00233=798156,0
EC00234=798156,0
EC00235=975524,0
EC00236=975524,0
EC00237=975524,0
EC00238=975524,0
EC00239=975524,0
EC00240=975524,0
EC00241=975524,0
EC00242=975524,0
EC00243=975524,0
EC00244=975524,0
EC00245=975524,0
EC00246=975524,0
EC00247=975524,0
EC00248=975524,0
EC00249=975524,0
EC00250=975524,0
EC00251=975524,0
EC00252=975524,0
EC00253=975524,0
EC00254=975524,0
EC00255=975524,0
EC00256=975524,0
EC00257=975524,0
EC00258=975524,0
EC00259=975524,0
EC00260=975524,0
EC00261=975524,0
EC00262=975524,0
EC00263=975524,0
EC00264=975524,0
EC00265=975524,0
EC00266=975524,0
EC00267=975524,0
EC00268=975524,0
EC00269=975524,0
EC00270=975524,0
EC00271=975524,0
EC00272=975524,0
EC00273=975524,0
EC00274=975524,0
EC00275=975524,0
EC00276=975524,0
EC00277=975524,0
EC00278=975524,0
EC00279=975524,0
EC00280=975524,0
EC00281=975524,0
EC00282=975524,0
EC00283=975524,0
EC00284=975524,0
EC00285=975524,0
EC00286=975524,0
EC00287=975524,0
EC00288=975524,0
EC00289=975524,0
EC00290=975524,0
EC00291=975524,0
EC00292=975524,0
EC00293=975524,0
EC00294=975524,0
EC00295=975524,0
EC00296=975524,0
EC00297=975524,0
EC00298=975524,0
EC00299=975524,0
EC00300=975524,0
EC00301=975524,0
EC00302=975524,0
EC00303=975524,0
EC00304=975524,0
EC00305=975524,0
EC00306=975524,0
EC00307=975524,0
EC00308=975524,0
EC00309=975524,0
EC00310=975524,0
EC00311=975524,0
EC00312=975524,0
EC00313=975524,0
EC00314=975524,0
EC00315=975524,0
EC00316=975524,0
EC00317=975524,0
EC00318=975524,0
EC00319=975524,0
EC00320=975524,0
EC00321=975524,0
EC00322=975524,0
EC00323=975524,0
EC00324=975524,0
EC00325=975524,0
EC00326=975524,0
EC00327=975524,0
EC00328=975524,0
EC00329=975524,0
EC00330=975524,0
EC00331=975524,0
EC00332=975524,0
EC00333=975524,0
EC00334=975524,0
EC00335=975524,0
EC00336=975524,0
EC00337=975524,0
EC00338=975524,0
EC00339=975524,0
EC00340=975524,0
EC00341=975524,0
EC00342=975524,0
EC00343=975524,0
EC00344=975524,0
EC00345=975524,0
EC00346=975524,0
EC00347=975524,0
EC00348=975524,0
EC00349=975524,0
EC00350=975524,0
EC00351=975524,0
EC00352=975524,0
EC00353=975524,0
EC00354=975524,0
EC00355=975524,0
EC00356=975524,0
EC00357=975524,0
EC00358=975524,0
EC00359=975524,0
EC00360=975524,0
EC00361=975524,0
EC00362=975524,0
EC00363=975524,0
EC00364=975524,0
EC00365=975524,0
EC00366=975524,0
EC00367=975524,0
EC00368=975524,0
EC00369=975524,0
EC00370=975524,0
EC00371=975524,0
EC00372=975524,0
EC00373=975524,0
EC00374=975524,0
EC00375=975524,0
EC00376=975524,0
EC00377=975524,0
EC00378=975522,1
EC00379=975524,0
EC00380=975524,0
EC00381=975524,0
EC00382=975524,0
EC00383=975524,0
EC00384=975524,0
EC00385=975524,0
EC00386=975524,0
EC00387=975524,0
EC00388=975524,0
EC00389=975524,0
EC00390=975524,0
EC00391=975524,0
EC00392=975524,0
EC00393=975524,0
EC00394=975524,0
EC00395=975524,0
EC00396=975524,0
EC00397=975524,0
EC00398=975524,0
EC00399=975524,0
EC00400=975524,0
EC00401=975524,0
EC00402=975524,0
EC00403=975524,0
EC00404=975524,0
EC00405=975524,0
EC00406=975524,0
EC00407=975524,0
EC00408=975524,0
EC00409=975524,0
EC00410=975522,1
EC00411=975524,0
EC00412=975524,0
EC00413=975524,0
EC00414=975524,0
EC00415=975524,0
EC00416=975524,0
EC00417=798156,0
EC00418=798156,0
EC00419=798156,0
EC00420=798156,0
EC00421=798156,0
EC00422=798156,0
EC00423=798156,0
EC00424=798156,0
EC00425=798156,0
EC00426=798156,0
EC00427=798156,0
EC00428=798156,0
EC00429=798156,0
EC00430=798156,0
EC00431=798156,0
EC00432=798156,0
EC00433=798156,0
EC00434=798156,0
EC00435=798156,0
EC00436=798156,0
EC00437=798156,0
EC00438=798156,0
EC00439=798156,0
EC00440=798156,0
EC00441=798156,0
EC00442=798156,0
EC00443=798156,0
EC00444=798156,0
EC00445=798156,0
EC00446=798156,0
EC00447=798156,0
EC00448=798156,0
EC00449=798156,0
EC00450=798156,0
EC00451=798156,0
EC00452=798156,0
EC00453=798156,0
EC00454=798156,0
EC00455=798156,0
EC00456=798156,0
EC00457=798156,0
EC00458=798156,0
EC00459=798156,0
EC00460=798156,0
EC00461=798156,0
EC00462=798156,0
EC00463=798156,0
EC00464=798156,0
EC00465=798156,0
EC00466=798156,0
EC00467=798156,0
EC00468=798156,0
EC00469=798156,0
EC00470=798156,0
EC00471=798156,0
EC00472=798156,0
EC00473=798156,0
EC00474=798156,0
EC00475=798156,0
EC00476=798156,0
EC00477=798156,0
EC00478=798156,0
EC00479=798156,0
EC00480=798156,0
EC00481=798156,0
EC00482=798156,0
EC00483=798156,0
EC00484=798156,0
EC00485=798156,0
EC00486=798156,0
EC00487=798156,0
EC00488=798156,0
EC00489=798156,0
EC00490=798156,0
EC00491=798156,0
EC00492=798156,0
EC00493=798156,0
EC00494=798156,0
EC00495=798156,0
EC00496=798156,0
EC00497=798156,0
EC00498=798156,0
EC00499=798156,0
EC00500=798156,0
EC00501=798156,0
EC00502=798156,0
EC00503=798156,0
EC00504=798156,0
EC00505=798156,0
EC00506=798156,0
EC00507=798156,0
EC00508=798156,0
EC00509=798156,0
EC00510=798156,0
EC00511=798156,0
EC00512=798156,0
EC00513=798156,0
EC00514=798147,5
EC00515=798147,5
EC00516=798147,5
EC00517=798147,5
EC00518=798147,5
EC00519=798147,5
EC00520=798147,5
EC00521=798147,5
EC00522=798147,5
EC00523=798147,5
EC00524=798147,5
EC00525=798147,5
EC00526=798147,5
EC00527=798147,5
EC00528=798147,5
EC00529=798147,5
EC00530=798147,5
EC00531=798147,5
EC00532=798147,5
EC00533=798147,5
EC00534=798147,5
EC00535=798147,5
EC00536=798147,5
EC00537=798147,5
EC00538=798147,5
EC00539=798147,5
EC00540=798147,5
EC00541=798147,5
EC00542=798147,5
EC00543=798147,5
EC00544=798147,5
EC00545=798147,5
EC00546=798147,5
EC00547=798147,5
EC00548=798147,5
EC00549=798147,5
EC00550=798147,5
EC00551=798147,5
EC00552=798146,6
EC00553=798146,6
EC00554=798146,6
EC00555=798146,6
EC00556=798146,6
EC00557=798146,6
EC00558=798146,6
EC00559=798146,6
EC00560=798146,6
EC00561=798146,6
EC00562=798146,6
EC00563=798146,6
EC00564=798146,6
EC00565=798146,6
EC00566=798146,6
EC00567=798146,6
EC00568=798146,6
EC00569=798146,6
EC00570=798146,6
EC00571=798146,6
EC00572=798146,6
EC00573=798146,6
EC00574=798146,6
///POSTYPE BASE
///RECTAN
///RCONF 0,0,0,0,0,0,0,0,0,0,0,0,0,0,0,0,0,0,0,0,0,0,0,0
P00006=0.222,-3.123,-1.508,0.0000,0.0000,0.0000
P00020=2.715,4.999,8.452,0.0000,0.0000,0.0000
P00021=-0.225,-6.128,-0.405,0.0000,0.0000,0.0000
P00022=0.222,-3.123,-1.508,0.0000,0.0000,0.0000
P00023=0.143,-0.036,0.682,0.0000,0.0000,0.0000
P00024=0.145,-0.552,1.326,0.0000,0.0000,0.0000
P00025=-2.003,0.006,0.728,0.0000,0.0000,0.0000
P00026=0.562,-0.002,-0.337,0.0000,0.0000,0.0000
P00031=1.853,-0.001,-1.549,0.0000,0.0000,0.0000
P00032=1.957,0.503,-7.217,0.0000,0.0000,0.0000
///RCONF 0,0,0,0,1,0,0,0,0,0,0,0,0,0,0,0,0,0,0,0,0,0,0,0
P00033=-0.123,0.612,-5.012,0.0000,0.0000,0.0000
///RCONF 0,0,0,0,0,0,0,0,0,0,0,0,0,0,0,0,0,0,0,0,0,0,0,0
P00034=-0.304,0.773,-2.693,0.0000,0.0000,0.0000
P00035=2.817,0.591,-1.622,0.0000,0.0000,0.0000
P00036=-1.108,-0.829,1.850,0.0000,0.0000,0.0000
P00037=0.023,0.937,-2.677,0.0000,0.0000,0.0000
P00038=0.158,-1.133,-1.952,0.0000,0.0000,0.0000
P00039=0.012,-3.081,-0.106,0.0000,0.0000,0.0000
P00040=-0.030,9.648,2.467,0.0000,0.0000,0.0000
P00041=0.192,3.924,0.305,0.0000,0.0000,0.0000
P00042=-0.217,1.941,0.413,0.0000,0.0000,0.0000
P00043=-0.044,-1.937,1.197,0.0000,0.0000,0.0000
P00044=0.687,-2.322,1.156,0.0000,0.0000,0.0000
P00045=-0.068,-0.810,1.603,0.0000,0.0000,0.0000
P00046=0.799,0.043,1.292,0.0000,0.0000,0.0000
///RCONF 0,1,0,0,0,0,0,0,0,0,0,0,0,0,0,0,0,0,0,0,0,0,0,0
P00047=-0.011,1.737,-0.646,0.0000,0.0000,0.0000
///RCONF 0,0,0,0,0,0,0,0,0,0,0,0,0,0,0,0,0,0,0,0,0,0,0,0
P00048=2.411,0.025,-0.606,0.0000,0.0000,0.0000
P00049=3.413,-3.572,-1.618,0.0000,0.0000,0.0000
P00050=4.296,-4.501,-0.826,0.0000,0.0000,0.0000
P00051=0.367,3.892,0.009,0.0000,0.0000,0.0000
P00052=0.088,2.832,-0.342,0.0000,0.0000,0.0000
P00053=0.134,6.594,0.107,0.0000,0.0000,0.0000
P00054=-0.103,6.509,-0.702,0.0000,0.0000,0.0000
P00055=-0.342,8.912,1.324,0.0000,0.0000,0.0000
P00056=0.568,-0.032,0.830,0.0000,0.0000,0.0000
P00057=0.586,-0.180,1.727,0.0000,0.0000,0.0000
P00058=0.385,-0.061,1.027,0.0000,0.0000,0.0000
//INST
///DATE 2025/03/12 14:06
///ATTR SC,RW
///GROUP1 RB1,BS1
///GROUP2 ST1
NOP
'X2_57-69(1)(90,0)
'Down
'Down
MOVJ C00000 BC00000 VJ=100.00  +MOVJ EC00000 VJ=100.00
MOVJ C00001 BC00001 VJ=100.00  +MOVJ EC00001 VJ=100.00
MOVJ C00002 BC00002 VJ=100.00  +MOVJ EC00002 VJ=100.00
'Path S4672
SFTOF3D
MOVJ C00003 BC00003 VJ=100.00  +MOVJ EC00003 VJ=100.00
MOVL C00004 BC00004 V=800.0  +MOVJ EC00004 VJ=100.00
SMOVL C00005 BC00005 V=166.7  +MOVJ EC00005
SREFP 3 C00006 BC00006  +REFP EC00006
CALL JOB:SEARCH-R1-S13D
SET P020 P006
SFTON3D P020
SMOVL C00007 BC00007 V=166.7  +MOVJ EC00007
SREFP 3 C00008 BC00008  +REFP EC00008
CALL JOB:SEARCH-R1-S13D
SET P020 P006
SFTON3D P020
SMOVL C00009 BC00009 V=166.7  +MOVJ EC00009
MOVL C00010 BC00010 V=800.0  +MOVJ EC00010 VJ=100.00
MOVL C00011 BC00011 V=1000.0  +MOVJ EC00011 VJ=100.00
'EndPath S4672
'Path S4673
SFTOF3D
MOVJ C00012 BC00012 VJ=100.00  +MOVJ EC00012 VJ=100.00
MOVJ C00013 BC00013 VJ=100.00  +MOVJ EC00013 VJ=100.00
MOVL C00014 BC00014 V=800.0  +MOVJ EC00014 VJ=100.00
SMOVL C00015 BC00015 V=166.7  +MOVJ EC00015
SREFP 3 C00016 BC00016  +REFP EC00016
CALL JOB:SEARCH-R1-S13D
SET P021 P006
SFTON3D P021
SMOVL C00017 BC00017 V=166.7  +MOVJ EC00017
SREFP 3 C00018 BC00018  +REFP EC00018
CALL JOB:SEARCH-R1-S13D
SET P021 P006
SFTON3D P021
SMOVL C00019 BC00019 V=166.7  +MOVJ EC00019
MOVL C00020 BC00020 V=800.0  +MOVJ EC00020 VJ=100.00
MOVL C00021 BC00021 V=1000.0  +MOVJ EC00021 VJ=100.00
'EndPath S4673
'Path S4674
SFTOF3D
MOVJ C00022 BC00022 VJ=100.00  +MOVJ EC00022 VJ=100.00
MOVL C00023 BC00023 V=800.0  +MOVJ EC00023 VJ=100.00
SMOVL C00024 BC00024 V=166.7  +MOVJ EC00024
SREFP 3 C00025 BC00025  +REFP EC00025
CALL JOB:SEARCH-R1-S13D
SET P022 P006
SFTON3D P022
SMOVL C00026 BC00026 V=166.7  +MOVJ EC00026
SMOVL C00027 BC00027 V=166.7  +MOVJ EC00027
SREFP 3 C00028 BC00028  +REFP EC00028
CALL JOB:SEARCH-R1-S13D
SET P022 P006
SFTON3D P022
SMOVL C00029 BC00029 V=166.7  +MOVJ EC00029
MOVL C00030 BC00030 V=800.0  +MOVJ EC00030 VJ=100.00
MOVL C00031 BC00031 V=1000.0  +MOVJ EC00031 VJ=100.00
'EndPath S4674
MOVJ C00032 BC00032 VJ=100.00  +MOVJ EC00032 VJ=100.00
MOVJ C00033 BC00033 VJ=100.00  +MOVJ EC00033 VJ=100.00
MOVJ C00034 BC00034 VJ=100.00  +MOVJ EC00034 VJ=100.00
MOVJ C00035 BC00035 VJ=100.00  +MOVJ EC00035 VJ=100.00
SFTOF3D
MOVJ C00036 BC00036 VJ=100.00  +MOVJ EC00036 VJ=100.00
SMOVL C00037 BC00037 V=166.7  +MOVJ EC00037
SREFP 3 C00038 BC00038  +REFP EC00038
CALL JOB:SEARCH-R1-S13D
SET P041 P006
SFTON3D P041
SMOVL C00039 BC00039 V=166.7  +MOVJ EC00039
SREFP 3 C00040 BC00040  +REFP EC00040
CALL JOB:SEARCH-R1-S13D
SET P041 P006
SFTON3D P041
SMOVL C00041 BC00041 V=166.7  +MOVJ EC00041
SMOVL C00042 BC00042 V=166.7  +MOVJ EC00042
SMOVL C00043 BC00043 V=166.7  +MOVJ EC00043
SREFP 3 C00044 BC00044  +REFP EC00044
CALL JOB:SEARCH-R1-S13D
SET P041 P006
SFTON3D P041
SMOVL C00045 BC00045 V=166.7  +MOVJ EC00045
SFTOF3D
MOVJ C00046 BC00046 VJ=100.00  +MOVJ EC00046 VJ=100.00
MOVL C00047 BC00047 V=800.0  +MOVJ EC00047 VJ=100.00
SMOVL C00048 BC00048 V=166.7  +MOVJ EC00048
SREFP 3 C00049 BC00049  +REFP EC00049
CALL JOB:SEARCH-R1-S13D
SET P042 P006
SFTON3D P042
SMOVL C00050 BC00050 V=166.7  +MOVJ EC00050
SREFP 3 C00051 BC00051  +REFP EC00051
CALL JOB:SEARCH-R1-S13D
SET P042 P006
SFTON3D P042
SMOVL C00052 BC00052 V=166.7  +MOVJ EC00052
SFTOF3D
MOVL C00053 BC00053 V=800.0  +MOVJ EC00053 VJ=100.00
SMOVL C00054 BC00054 V=166.7  +MOVJ EC00054
SREFP 3 C00055 BC00055  +REFP EC00055
CALL JOB:SEARCH-R1-S13D
SET P043 P006
SFTON3D P043
SMOVL C00056 BC00056 V=166.7  +MOVJ EC00056
SREFP 3 C00057 BC00057  +REFP EC00057
CALL JOB:SEARCH-R1-S13D
SET P043 P006
SFTON3D P043
SMOVL C00058 BC00058 V=166.7  +MOVJ EC00058
SMOVL C00059 BC00059 V=166.7  +MOVJ EC00059
MOVJ C00060 BC00060 VJ=100.00  +MOVJ EC00060 VJ=100.00
MOVJ C00061 BC00061 VJ=100.00  +MOVJ EC00061 VJ=100.00
MOVJ C00062 BC00062 VJ=100.00  +MOVJ EC00062 VJ=100.00
MOVJ C00063 BC00063 VJ=100.00  +MOVJ EC00063 VJ=100.00
MOVJ C00064 BC00064 VJ=100.00  +MOVJ EC00064 VJ=100.00
SMOVL C00065 BC00065 V=166.7  +MOVJ EC00065
SREFP 3 C00066 BC00066  +REFP EC00066
CALL JOB:SEARCH-R1-S13D
SET P044 P006
SFTON3D P044
SMOVL C00067 BC00067 V=166.7  +MOVJ EC00067
SREFP 3 C00068 BC00068  +REFP EC00068
CALL JOB:SEARCH-R1-S13D
SET P044 P006
SFTON3D P044
SMOVL C00069 BC00069 V=166.7  +MOVJ EC00069
SREFP 3 C00070 BC00070  +REFP EC00070
CALL JOB:SEARCH-R1-S13D
SET P044 P006
SFTON3D P044
SMOVL C00071 BC00071 V=166.7  +MOVJ EC00071
SMOVL C00072 BC00072 V=166.7  +MOVJ EC00072
SREFP 3 C00073 BC00073  +REFP EC00073
CALL JOB:SEARCH-R1-S13D
SET P045 P006
SFTON3D P045
SMOVL C00074 BC00074 V=166.7  +MOVJ EC00074
SREFP 3 C00075 BC00075  +REFP EC00075
CALL JOB:SEARCH-R1-S13D
SET P045 P006
SFTON3D P045
SMOVL C00076 BC00076 V=166.7  +MOVJ EC00076
SREFP 3 C00077 BC00077  +REFP EC00077
CALL JOB:SEARCH-R1-S13D
SET P045 P006
SFTON3D P045
SMOVL C00078 BC00078 V=166.7  +MOVJ EC00078
MOVL C00079 BC00079 V=666.7  +MOVJ EC00079 VJ=100.00
MOVL C00080 BC00080 V=1000.0  +MOVJ EC00080 VJ=100.00
SMOVL C00081 BC00081 V=166.7  +MOVJ EC00081
SREFP 3 C00082 BC00082  +REFP EC00082
CALL JOB:SEARCH-R1-S13D
SET P046 P006
SFTON3D P046
SMOVL C00083 BC00083 V=166.7  +MOVJ EC00083
SREFP 3 C00084 BC00084  +REFP EC00084
CALL JOB:SEARCH-R1-S13D
SET P046 P006
SFTON3D P046
SMOVL C00085 BC00085 V=166.7  +MOVJ EC00085
SMOVL C00086 BC00086 V=166.7  +MOVJ EC00086
SREFP 3 C00087 BC00087  +REFP EC00087
CALL JOB:SEARCH-R1-S13D
SET P046 P006
SFTON3D P046
SMOVL C00088 BC00088 V=166.7  +MOVJ EC00088
MOVL C00089 BC00089 V=166.7  +MOVJ EC00089 VJ=100.00
SMOVL C00090 BC00090 V=166.7  +MOVJ EC00090
SREFP 3 C00091 BC00091  +REFP EC00091
CALL JOB:SEARCH-R1-S13D
SET P047 P006
SFTON3D P047
SMOVL C00092 BC00092 V=166.7  +MOVJ EC00092
SREFP 3 C00093 BC00093  +REFP EC00093
CALL JOB:SEARCH-R1-S13D
SET P047 P006
SFTON3D P047
SMOVL C00094 BC00094 V=166.7  +MOVJ EC00094
SMOVL C00095 BC00095 V=166.7  +MOVJ EC00095
SREFP 3 C00096 BC00096  +REFP EC00096
CALL JOB:SEARCH-R1-S13D
SET P047 P006
SFTON3D P047
SMOVL C00097 BC00097 V=166.7  +MOVJ EC00097
SMOVL C00098 BC00098 V=1000.0  +MOVJ EC00098
SMOVL C00099 BC00099 V=166.7  +MOVJ EC00099
SREFP 3 C00100 BC00100  +REFP EC00100
CALL JOB:SEARCH-R1-S13D
SET P048 P006
SFTON3D P048
SMOVL C00101 BC00101 V=166.7  +MOVJ EC00101
SREFP 3 C00102 BC00102  +REFP EC00102
CALL JOB:SEARCH-R1-S13D
SET P048 P006
SFTON3D P048
SMOVL C00103 BC00103 V=166.7  +MOVJ EC00103
SMOVL C00104 BC00104 V=166.7  +MOVJ EC00104
SREFP 3 C00105 BC00105  +REFP EC00105
CALL JOB:SEARCH-R1-S13D
SET P048 P006
SFTON3D P048
SMOVL C00106 BC00106 V=166.7  +MOVJ EC00106
SMOVL C00107 BC00107 V=166.7  +MOVJ EC00107
SREFP 3 C00108 BC00108  +REFP EC00108
CALL JOB:SEARCH-R1-S13D
SET P049 P006
SFTON3D P049
SMOVL C00109 BC00109 V=166.7  +MOVJ EC00109
SREFP 3 C00110 BC00110  +REFP EC00110
CALL JOB:SEARCH-R1-S13D
SET P049 P006
SFTON3D P049
SMOVL C00111 BC00111 V=166.7  +MOVJ EC00111
SMOVL C00112 BC00112 V=166.7  +MOVJ EC00112
SREFP 3 C00113 BC00113  +REFP EC00113
CALL JOB:SEARCH-R1-S13D
SET P049 P006
SFTON3D P049
SMOVL C00114 BC00114 V=166.7  +MOVJ EC00114
SFTOF3D
SMOVL C00115 BC00115 V=1000.0  +MOVJ EC00115
SMOVL C00116 BC00116 V=1000.0  +MOVJ EC00116
SMOVL C00117 BC00117 V=166.7  +MOVJ EC00117
SREFP 3 C00118 BC00118  +REFP EC00118
CALL JOB:SEARCH-R1-S13D
SET P050 P006
SFTON3D P050
SMOVL C00119 BC00119 V=166.7  +MOVJ EC00119
SMOVL C00120 BC00120 V=166.7  +MOVJ EC00120
SMOVL C00121 BC00121 V=166.7  +MOVJ EC00121
SREFP 3 C00122 BC00122  +REFP EC00122
CALL JOB:SEARCH-R1-S13D
SET P050 P006
SFTON3D P050
SMOVL C00123 BC00123 V=166.7  +MOVJ EC00123
SFTOF3D
SMOVL C00124 BC00124 V=666.7  +MOVJ EC00124
SMOVL C00125 BC00125 V=166.7  +MOVJ EC00125
SREFP 3 C00126 BC00126  +REFP EC00126
CALL JOB:SEARCH-R1-S13D
SET P051 P006
SFTON3D P051
SMOVL C00127 BC00127 V=166.7  +MOVJ EC00127
SMOVL C00128 BC00128 V=166.7  +MOVJ EC00128
SMOVL C00129 BC00129 V=166.7  +MOVJ EC00129
SREFP 3 C00130 BC00130  +REFP EC00130
CALL JOB:SEARCH-R1-S13D
SET P051 P006
SFTON3D P051
SMOVL C00131 BC00131 V=166.7  +MOVJ EC00131
SFTOF3D
SMOVL C00132 BC00132 V=666.7  +MOVJ EC00132
SMOVL C00133 BC00133 V=166.7  +MOVJ EC00133
SREFP 3 C00134 BC00134  +REFP EC00134
CALL JOB:SEARCH-R1-S13D
SET P052 P006
SFTON3D P052
SMOVL C00135 BC00135 V=166.7  +MOVJ EC00135
SMOVL C00136 BC00136 V=166.7  +MOVJ EC00136
SMOVL C00137 BC00137 V=166.7  +MOVJ EC00137
SREFP 3 C00138 BC00138  +REFP EC00138
CALL JOB:SEARCH-R1-S13D
SET P052 P006
SFTON3D P052
SMOVL C00139 BC00139 V=166.7  +MOVJ EC00139
SFTOF3D
SMOVL C00140 BC00140 V=666.7  +MOVJ EC00140
SMOVL C00141 BC00141 V=666.7  +MOVJ EC00141
SMOVL C00142 BC00142 V=166.7  +MOVJ EC00142
SREFP 3 C00143 BC00143  +REFP EC00143
CALL JOB:SEARCH-R1-S13D
SET P053 P006
SFTON3D P053
SMOVL C00144 BC00144 V=166.7  +MOVJ EC00144
SREFP 3 C00145 BC00145  +REFP EC00145
CALL JOB:SEARCH-R1-S13D
SET P053 P006
SFTON3D P053
SMOVL C00146 BC00146 V=166.7  +MOVJ EC00146
SMOVL C00147 BC00147 V=166.7  +MOVJ EC00147
SREFP 3 C00148 BC00148  +REFP EC00148
CALL JOB:SEARCH-R1-S13D
SET P053 P006
SFTON3D P053
SMOVL C00149 BC00149 V=166.7  +MOVJ EC00149
SMOVL C00150 BC00150 V=166.7  +MOVJ EC00150
SREFP 3 C00151 BC00151  +REFP EC00151
CALL JOB:SEARCH-R1-S13D
SET P054 P006
SFTON3D P054
SMOVL C00152 BC00152 V=166.7  +MOVJ EC00152
SREFP 3 C00153 BC00153  +REFP EC00153
CALL JOB:SEARCH-R1-S13D
SET P054 P006
SFTON3D P054
SMOVL C00154 BC00154 V=166.7  +MOVJ EC00154
SMOVL C00155 BC00155 V=166.7  +MOVJ EC00155
SREFP 3 C00156 BC00156  +REFP EC00156
CALL JOB:SEARCH-R1-S13D
SET P054 P006
SFTON3D P054
SMOVL C00157 BC00157 V=166.7  +MOVJ EC00157
SMOVL C00158 BC00158 V=666.7  +MOVJ EC00158
SMOVL C00159 BC00159 V=166.7  +MOVJ EC00159
SREFP 3 C00160 BC00160  +REFP EC00160
CALL JOB:SEARCH-R1-S13D
SET P055 P006
SFTON3D P055
SMOVL C00161 BC00161 V=166.7  +MOVJ EC00161
SREFP 3 C00162 BC00162  +REFP EC00162
CALL JOB:SEARCH-R1-S13D
SET P055 P006
SFTON3D P055
SMOVL C00163 BC00163 V=166.7  +MOVJ EC00163
SMOVL C00164 BC00164 V=166.7  +MOVJ EC00164
SREFP 3 C00165 BC00165  +REFP EC00165
CALL JOB:SEARCH-R1-S13D
SET P055 P006
SFTON3D P055
SMOVL C00166 BC00166 V=166.7  +MOVJ EC00166
SMOVL C00167 BC00167 V=166.7  +MOVJ EC00167
SREFP 3 C00168 BC00168  +REFP EC00168
CALL JOB:SEARCH-R1-S13D
SET P056 P006
SFTON3D P056
SMOVL C00169 BC00169 V=166.7  +MOVJ EC00169
SREFP 3 C00170 BC00170  +REFP EC00170
CALL JOB:SEARCH-R1-S13D
SET P056 P006
SFTON3D P056
SMOVL C00171 BC00171 V=166.7  +MOVJ EC00171
SMOVL C00172 BC00172 V=166.7  +MOVJ EC00172
SREFP 3 C00173 BC00173  +REFP EC00173
CALL JOB:SEARCH-R1-S13D
SET P056 P006
SFTON3D P056
SMOVL C00174 BC00174 V=166.7  +MOVJ EC00174
SMOVL C00175 BC00175 V=666.7  +MOVJ EC00175
SMOVL C00176 BC00176 V=666.7  +MOVJ EC00176
SMOVL C00177 BC00177 V=166.7  +MOVJ EC00177
SREFP 3 C00178 BC00178  +REFP EC00178
CALL JOB:SEARCH-R1-S13D
SET P057 P006
SFTON3D P057
SMOVL C00179 BC00179 V=166.7  +MOVJ EC00179
SREFP 3 C00180 BC00180  +REFP EC00180
CALL JOB:SEARCH-R1-S13D
SET P057 P006
SFTON3D P057
SMOVL C00181 BC00181 V=166.7  +MOVJ EC00181
SMOVL C00182 BC00182 V=166.7  +MOVJ EC00182
SREFP 3 C00183 BC00183  +REFP EC00183
CALL JOB:SEARCH-R1-S13D
SET P057 P006
SFTON3D P057
SMOVL C00184 BC00184 V=166.7  +MOVJ EC00184
SMOVL C00185 BC00185 V=166.7  +MOVJ EC00185
SREFP 3 C00186 BC00186  +REFP EC00186
CALL JOB:SEARCH-R1-S13D
SET P058 P006
SFTON3D P058
SMOVL C00187 BC00187 V=166.7  +MOVJ EC00187
SREFP 3 C00188 BC00188  +REFP EC00188
CALL JOB:SEARCH-R1-S13D
SET P058 P006
SFTON3D P058
SMOVL C00189 BC00189 V=166.7  +MOVJ EC00189
SMOVL C00190 BC00190 V=166.7  +MOVJ EC00190
SREFP 3 C00191 BC00191  +REFP EC00191
CALL JOB:SEARCH-R1-S13D
SET P058 P006
SFTON3D P058
SMOVL C00192 BC00192 V=166.7  +MOVJ EC00192
SFTOF3D
MOVL C00193 BC00193 V=666.7  +MOVJ EC00193 VJ=100.00
MOVJ C00194 BC00194 VJ=100.00  +MOVJ EC00194 VJ=100.00
MOVJ C00195 BC00195 VJ=100.00  +MOVJ EC00195 VJ=100.00
'Path S4677
SFTOF3D
MOVJ C00196 BC00196 VJ=100.00  +MOVJ EC00196 VJ=100.00
MOVL C00197 BC00197 V=800.0  +MOVJ EC00197 VJ=100.00
SMOVL C00198 BC00198 V=166.7  +MOVJ EC00198
SREFP 3 C00199 BC00199  +REFP EC00199
CALL JOB:SEARCH-R1-S13D
SET P023 P006
SFTON3D P023
SMOVL C00200 BC00200 V=166.7  +MOVJ EC00200
SREFP 3 C00201 BC00201  +REFP EC00201
CALL JOB:SEARCH-R1-S13D
SET P023 P006
SFTON3D P023
SMOVL C00202 BC00202 V=166.7  +MOVJ EC00202
SMOVL C00203 BC00203 V=166.7  +MOVJ EC00203
SREFP 3 C00204 BC00204  +REFP EC00204
CALL JOB:SEARCH-R1-S13D
SET P023 P006
SFTON3D P023
SMOVL C00205 BC00205 V=166.7  +MOVJ EC00205
MOVL C00206 BC00206 V=1000.0  +MOVJ EC00206 VJ=100.00
'EndPath S4677
'Path S4678
SFTOF3D
MOVJ C00207 BC00207 VJ=100.00  +MOVJ EC00207 VJ=100.00
MOVL C00208 BC00208 V=800.0  +MOVJ EC00208 VJ=100.00
SMOVL C00209 BC00209 V=166.7  +MOVJ EC00209
SREFP 3 C00210 BC00210  +REFP EC00210
CALL JOB:SEARCH-R1-S13D
SET P024 P006
SFTON3D P024
SMOVL C00211 BC00211 V=166.7  +MOVJ EC00211
SREFP 3 C00212 BC00212  +REFP EC00212
CALL JOB:SEARCH-R1-S13D
SET P024 P006
SFTON3D P024
SMOVL C00213 BC00213 V=166.7  +MOVJ EC00213
MOVL C00214 BC00214 V=1000.0  +MOVJ EC00214 VJ=100.00
'EndPath S4678
MOVJ C00215 BC00215 VJ=100.00  +MOVJ EC00215 VJ=100.00
MOVJ C00216 BC00216 VJ=100.00  +MOVJ EC00216 VJ=100.00
'Path S4679
SFTOF3D
MOVJ C00217 BC00217 VJ=100.00  +MOVJ EC00217 VJ=100.00
MOVL C00218 BC00218 V=800.0  +MOVJ EC00218 VJ=100.00
SMOVL C00219 BC00219 V=166.7  +MOVJ EC00219
SREFP 3 C00220 BC00220  +REFP EC00220
CALL JOB:SEARCH-R1-S13D
SET P025 P006
SFTON3D P025
SMOVL C00221 BC00221 V=166.7  +MOVJ EC00221
SREFP 3 C00222 BC00222  +REFP EC00222
CALL JOB:SEARCH-R1-S13D
SET P025 P006
SFTON3D P025
SMOVL C00223 BC00223 V=166.7  +MOVJ EC00223
MOVL C00224 BC00224 V=1000.0  +MOVJ EC00224 VJ=100.00
'EndPath S4679
'Path S4680
SFTOF3D
MOVJ C00225 BC00225 VJ=100.00  +MOVJ EC00225 VJ=100.00
MOVL C00226 BC00226 V=800.0  +MOVJ EC00226 VJ=100.00
SMOVL C00227 BC00227 V=166.7  +MOVJ EC00227
SREFP 3 C00228 BC00228  +REFP EC00228
CALL JOB:SEARCH-R1-S13D
SET P026 P006
SFTON3D P026
SMOVL C00229 BC00229 V=166.7  +MOVJ EC00229
SMOVL C00230 BC00230 V=166.7  +MOVJ EC00230
SREFP 3 C00231 BC00231  +REFP EC00231
CALL JOB:SEARCH-R1-S13D
SET P026 P006
SFTON3D P026
SMOVL C00232 BC00232 V=166.7  +MOVJ EC00232
MOVL C00233 BC00233 V=1000.0  +MOVJ EC00233 VJ=100.00
'EndPath S4680
MOVJ C00234 BC00234 VJ=100.00  +MOVJ EC00234 VJ=100.00
'Up
MOVJ C00235 BC00235 VJ=100.00  +MOVJ EC00235 VJ=100.00
MOVJ C00236 BC00236 VJ=100.00  +MOVJ EC00236 VJ=100.00
'Path S4681
SFTOF3D
MOVJ C00237 BC00237 VJ=100.00  +MOVJ EC00237 VJ=100.00
MOVL C00238 BC00238 V=800.0  +MOVJ EC00238 VJ=100.00
SMOVL C00239 BC00239 V=166.7  +MOVJ EC00239
SREFP 3 C00240 BC00240  +REFP EC00240
CALL JOB:SEARCH-R1-S13D
SET P031 P006
SFTON3D P031
SMOVL C00241 BC00241 V=166.7  +MOVJ EC00241
SREFP 3 C00242 BC00242  +REFP EC00242
CALL JOB:SEARCH-R1-S13D
SET P031 P006
SFTON3D P031
SMOVL C00243 BC00243 V=166.7  +MOVJ EC00243
SMOVL C00244 BC00244 V=166.7  +MOVJ EC00244
SREFP 3 C00245 BC00245  +REFP EC00245
CALL JOB:SEARCH-R1-S13D
SET P031 P006
SFTON3D P031
SMOVL C00246 BC00246 V=166.7  +MOVJ EC00246
MOVL C00247 BC00247 V=800.0  +MOVJ EC00247 VJ=100.00
MOVL C00248 BC00248 V=1000.0  +MOVJ EC00248 VJ=100.00
'EndPath S4681
MOVJ C00249 BC00249 VJ=100.00  +MOVJ EC00249 VJ=100.00
'Path S4682
SFTOF3D
MOVJ C00250 BC00250 VJ=100.00  +MOVJ EC00250 VJ=100.00
MOVL C00251 BC00251 V=800.0  +MOVJ EC00251 VJ=100.00
SMOVL C00252 BC00252 V=166.7  +MOVJ EC00252
SREFP 3 C00253 BC00253  +REFP EC00253
CALL JOB:SEARCH-R1-S13D
SET P032 P006
SFTON3D P032
SMOVL C00254 BC00254 V=166.7  +MOVJ EC00254
SREFP 3 C00255 BC00255  +REFP EC00255
CALL JOB:SEARCH-R1-S13D
SET P032 P006
SFTON3D P032
SMOVL C00256 BC00256 V=166.7  +MOVJ EC00256
SMOVL C00257 BC00257 V=166.7  +MOVJ EC00257
SREFP 3 C00258 BC00258  +REFP EC00258
CALL JOB:SEARCH-R1-S13D
SET P032 P006
SFTON3D P032
SMOVL C00259 BC00259 V=166.7  +MOVJ EC00259
MOVL C00260 BC00260 V=1000.0  +MOVJ EC00260 VJ=100.00
'EndPath S4682
MOVJ C00261 BC00261 VJ=100.00  +MOVJ EC00261 VJ=100.00
'Path S4683
SFTOF3D
MOVJ C00262 BC00262 VJ=100.00  +MOVJ EC00262 VJ=100.00
MOVL C00263 BC00263 V=800.0  +MOVJ EC00263 VJ=100.00
SMOVL C00264 BC00264 V=166.7  +MOVJ EC00264
SREFP 3 C00265 BC00265  +REFP EC00265
CALL JOB:SEARCH-R1-S13D
SET P033 P006
SFTON3D P033
SMOVL C00266 BC00266 V=166.7  +MOVJ EC00266
SREFP 3 C00267 BC00267  +REFP EC00267
CALL JOB:SEARCH-R1-S13D
SET P033 P006
SFTON3D P033
SMOVL C00268 BC00268 V=166.7  +MOVJ EC00268
SMOVL C00269 BC00269 V=166.7  +MOVJ EC00269
SREFP 3 C00270 BC00270  +REFP EC00270
CALL JOB:SEARCH-R1-S13D
SET P033 P006
SFTON3D P033
SMOVL C00271 BC00271 V=166.7  +MOVJ EC00271
MOVL C00272 BC00272 V=1000.0  +MOVJ EC00272 VJ=100.00
MOVL C00273 BC00273 V=1000.0  +MOVJ EC00273 VJ=100.00
'EndPath S4683
MOVJ C00274 BC00274 VJ=100.00  +MOVJ EC00274 VJ=100.00
'Path S4684
SFTOF3D
MOVJ C00275 BC00275 VJ=100.00  +MOVJ EC00275 VJ=100.00
MOVL C00276 BC00276 V=800.0  +MOVJ EC00276 VJ=100.00
SMOVL C00277 BC00277 V=166.7  +MOVJ EC00277
SREFP 3 C00278 BC00278  +REFP EC00278
CALL JOB:SEARCH-R1-S13D
SET P034 P006
SFTON3D P034
SMOVL C00279 BC00279 V=166.7  +MOVJ EC00279
SREFP 3 C00280 BC00280  +REFP EC00280
CALL JOB:SEARCH-R1-S13D
SET P034 P006
SFTON3D P034
SMOVL C00281 BC00281 V=166.7  +MOVJ EC00281
SMOVL C00282 BC00282 V=166.7  +MOVJ EC00282
SREFP 3 C00283 BC00283  +REFP EC00283
CALL JOB:SEARCH-R1-S13D
SET P034 P006
SFTON3D P034
SMOVL C00284 BC00284 V=166.7  +MOVJ EC00284
MOVL C00285 BC00285 V=800.0  +MOVJ EC00285 VJ=100.00
MOVL C00286 BC00286 V=1000.0  +MOVJ EC00286 VJ=100.00
MOVL C00287 BC00287 V=1000.0  +MOVJ EC00287 VJ=100.00
'EndPath S4684
MOVJ C00288 BC00288 VJ=100.00  +MOVJ EC00288 VJ=100.00
'Path S4685
SFTOF3D
MOVJ C00289 BC00289 VJ=100.00  +MOVJ EC00289 VJ=100.00
MOVL C00290 BC00290 V=800.0  +MOVJ EC00290 VJ=100.00
SMOVL C00291 BC00291 V=166.7  +MOVJ EC00291
SREFP 3 C00292 BC00292  +REFP EC00292
CALL JOB:SEARCH-R1-S13D
SET P035 P006
SFTON3D P035
SMOVL C00293 BC00293 V=166.7  +MOVJ EC00293
SMOVL C00294 BC00294 V=166.7  +MOVJ EC00294
SREFP 3 C00295 BC00295  +REFP EC00295
CALL JOB:SEARCH-R1-S13D
SET P035 P006
SFTON3D P035
SMOVL C00296 BC00296 V=166.7  +MOVJ EC00296
SMOVL C00297 BC00297 V=166.7  +MOVJ EC00297
SREFP 3 C00298 BC00298  +REFP EC00298
CALL JOB:SEARCH-R1-S13D
SET P035 P006
SFTON3D P035
SMOVL C00299 BC00299 V=166.7  +MOVJ EC00299
MOVL C00300 BC00300 V=1000.0  +MOVJ EC00300 VJ=100.00
'EndPath S4685
MOVJ C00301 BC00301 VJ=100.00  +MOVJ EC00301 VJ=100.00
'Path S4686
SFTOF3D
MOVJ C00302 BC00302 VJ=100.00  +MOVJ EC00302 VJ=100.00
MOVL C00303 BC00303 V=800.0  +MOVJ EC00303 VJ=100.00
SMOVL C00304 BC00304 V=166.7  +MOVJ EC00304
SREFP 3 C00305 BC00305  +REFP EC00305
CALL JOB:SEARCH-R1-S13D
SET P036 P006
SFTON3D P036
SMOVL C00306 BC00306 V=166.7  +MOVJ EC00306
SMOVL C00307 BC00307 V=166.7  +MOVJ EC00307
SREFP 3 C00308 BC00308  +REFP EC00308
CALL JOB:SEARCH-R1-S13D
SET P036 P006
SFTON3D P036
SMOVL C00309 BC00309 V=166.7  +MOVJ EC00309
SMOVL C00310 BC00310 V=166.7  +MOVJ EC00310
SREFP 3 C00311 BC00311  +REFP EC00311
CALL JOB:SEARCH-R1-S13D
SET P036 P006
SFTON3D P036
SMOVL C00312 BC00312 V=166.7  +MOVJ EC00312
MOVL C00313 BC00313 V=1000.0  +MOVJ EC00313 VJ=100.00
'EndPath S4686
MOVJ C00314 BC00314 VJ=100.00  +MOVJ EC00314 VJ=100.00
'Path S4687
SFTOF3D
MOVJ C00315 BC00315 VJ=100.00  +MOVJ EC00315 VJ=100.00
MOVL C00316 BC00316 V=800.0  +MOVJ EC00316 VJ=100.00
SMOVL C00317 BC00317 V=166.7  +MOVJ EC00317
SREFP 3 C00318 BC00318  +REFP EC00318
CALL JOB:SEARCH-R1-S13D
SET P037 P006
SFTON3D P037
SMOVL C00319 BC00319 V=166.7  +MOVJ EC00319
SMOVL C00320 BC00320 V=166.7  +MOVJ EC00320
SREFP 3 C00321 BC00321  +REFP EC00321
CALL JOB:SEARCH-R1-S13D
SET P037 P006
SFTON3D P037
SMOVL C00322 BC00322 V=166.7  +MOVJ EC00322
SMOVL C00323 BC00323 V=166.7  +MOVJ EC00323
SREFP 3 C00324 BC00324  +REFP EC00324
CALL JOB:SEARCH-R1-S13D
SET P037 P006
SFTON3D P037
SMOVL C00325 BC00325 V=166.7  +MOVJ EC00325
MOVL C00326 BC00326 V=1000.0  +MOVJ EC00326 VJ=100.00
'EndPath S4687
MOVJ C00327 BC00327 VJ=100.00  +MOVJ EC00327 VJ=100.00
'Path S4688
SFTOF3D
MOVJ C00328 BC00328 VJ=100.00  +MOVJ EC00328 VJ=100.00
MOVL C00329 BC00329 V=800.0  +MOVJ EC00329 VJ=100.00
SMOVL C00330 BC00330 V=166.7  +MOVJ EC00330
SREFP 3 C00331 BC00331  +REFP EC00331
CALL JOB:SEARCH-R1-S13D
SET P038 P006
SFTON3D P038
SMOVL C00332 BC00332 V=166.7  +MOVJ EC00332
SMOVL C00333 BC00333 V=166.7  +MOVJ EC00333
SREFP 3 C00334 BC00334  +REFP EC00334
CALL JOB:SEARCH-R1-S13D
SET P038 P006
SFTON3D P038
SMOVL C00335 BC00335 V=166.7  +MOVJ EC00335
SMOVL C00336 BC00336 V=166.7  +MOVJ EC00336
SREFP 3 C00337 BC00337  +REFP EC00337
CALL JOB:SEARCH-R1-S13D
SET P038 P006
SFTON3D P038
SMOVL C00338 BC00338 V=166.7  +MOVJ EC00338
MOVL C00339 BC00339 V=800.0  +MOVJ EC00339 VJ=100.00
MOVL C00340 BC00340 V=1000.0  +MOVJ EC00340 VJ=100.00
'EndPath S4688
MOVJ C00341 BC00341 VJ=100.00  +MOVJ EC00341 VJ=100.00
'Path S4689
SFTOF3D
MOVJ C00342 BC00342 VJ=100.00  +MOVJ EC00342 VJ=100.00
MOVL C00343 BC00343 V=800.0  +MOVJ EC00343 VJ=100.00
SMOVL C00344 BC00344 V=166.7  +MOVJ EC00344
SREFP 3 C00345 BC00345  +REFP EC00345
CALL JOB:SEARCH-R1-S13D
SET P039 P006
SFTON3D P039
SMOVL C00346 BC00346 V=166.7  +MOVJ EC00346
SMOVL C00347 BC00347 V=166.7  +MOVJ EC00347
SREFP 3 C00348 BC00348  +REFP EC00348
CALL JOB:SEARCH-R1-S13D
SET P039 P006
SFTON3D P039
SMOVL C00349 BC00349 V=166.7  +MOVJ EC00349
SMOVL C00350 BC00350 V=166.7  +MOVJ EC00350
SREFP 3 C00351 BC00351  +REFP EC00351
CALL JOB:SEARCH-R1-S13D
SET P039 P006
SFTON3D P039
SMOVL C00352 BC00352 V=166.7  +MOVJ EC00352
MOVL C00353 BC00353 V=1000.0  +MOVJ EC00353 VJ=100.00
'EndPath S4689
'Path S4690
SFTOF3D
MOVJ C00354 BC00354 VJ=100.00  +MOVJ EC00354 VJ=100.00
MOVL C00355 BC00355 V=800.0  +MOVJ EC00355 VJ=100.00
SMOVL C00356 BC00356 V=166.7  +MOVJ EC00356
SREFP 3 C00357 BC00357  +REFP EC00357
CALL JOB:SEARCH-R1-S13D
SET P040 P006
SFTON3D P040
SMOVL C00358 BC00358 V=166.7  +MOVJ EC00358
SREFP 3 C00359 BC00359  +REFP EC00359
CALL JOB:SEARCH-R1-S13D
SET P040 P006
SFTON3D P040
SMOVL C00360 BC00360 V=166.7  +MOVJ EC00360
MOVL C00361 BC00361 V=1000.0  +MOVJ EC00361 VJ=100.00
'EndPath S4690
'Path W4691
SFTOF3D
SFTON3D P039
MOVJ C00362 BC00362 VJ=100.00  +MOVJ EC00362 VJ=100.00
SMOVL C00363 BC00363 V=800.0  +MOVJ EC00363
SMOVL C00364 BC00364 V=166.7 PL=0  +MOVJ EC00364
MACRO1 MJ#(0) ARGF21
ARCON
SMOVL C00365 BC00365 V=7.5  +MOVJ EC00365
SFTON3D P040
SMOVL C00366 BC00366 V=7.5  +MOVJ EC00366
SMOVL C00367 BC00367 V=7.5  +MOVJ EC00367
ARCOF
SMOVL C00368 BC00368 V=800.0  +MOVJ EC00368
SMOVL C00369 BC00369 V=1000.0  +MOVJ EC00369
SFTOF3D
'EndPath W4691
'Path W4692
SFTOF3D
SFTON3D P037
MOVJ C00370 BC00370 VJ=100.00  +MOVJ EC00370 VJ=100.00
MOVJ C00371 BC00371 VJ=100.00  +MOVJ EC00371 VJ=100.00
MOVJ C00372 BC00372 VJ=100.00  +MOVJ EC00372 VJ=100.00
SMOVL C00373 BC00373 V=800.0  +MOVJ EC00373
SMOVL C00374 BC00374 V=166.7 PL=0  +MOVJ EC00374
MACRO1 MJ#(0) ARGF14
ARCON
SMOVL C00375 BC00375 V=10.0  +MOVJ EC00375
SMOVL C00376 BC00376 V=10.0  +MOVJ EC00376
SMOVL C00377 BC00377 V=10.0  +MOVJ EC00377
SFTON3D P038
SMOVL C00378 BC00378 V=10.0  +MOVJ EC00378
SMOVL C00379 BC00379 V=10.0  +MOVJ EC00379
ARCOF
SMOVL C00380 BC00380 V=800.0  +MOVJ EC00380
SMOVL C00381 BC00381 V=1000.0  +MOVJ EC00381
SFTOF3D
'EndPath W4692
MOVJ C00382 BC00382 VJ=100.00  +MOVJ EC00382 VJ=100.00
'Path W4693
SFTOF3D
SFTON3D P035
MOVJ C00383 BC00383 VJ=100.00  +MOVJ EC00383 VJ=100.00
MOVJ C00384 BC00384 VJ=100.00  +MOVJ EC00384 VJ=100.00
SMOVL C00385 BC00385 V=800.0  +MOVJ EC00385
SMOVL C00386 BC00386 V=166.7 PL=0  +MOVJ EC00386
ARCON
SMOVL C00387 BC00387 V=10.0  +MOVJ EC00387
SMOVL C00388 BC00388 V=10.0  +MOVJ EC00388
SMOVL C00389 BC00389 V=10.0  +MOVJ EC00389
SFTON3D P036
SMOVL C00390 BC00390 V=10.0  +MOVJ EC00390
SMOVL C00391 BC00391 V=10.0  +MOVJ EC00391
ARCOF
SMOVL C00392 BC00392 V=800.0  +MOVJ EC00392
SMOVL C00393 BC00393 V=1000.0  +MOVJ EC00393
SMOVL C00394 BC00394 V=1000.0  +MOVJ EC00394
SFTOF3D
'EndPath W4693
MOVJ C00395 BC00395 VJ=100.00  +MOVJ EC00395 VJ=100.00
'Path W4694
SFTOF3D
SFTON3D P033
MOVJ C00396 BC00396 VJ=100.00  +MOVJ EC00396 VJ=100.00
SMOVL C00397 BC00397 V=800.0  +MOVJ EC00397
SMOVL C00398 BC00398 V=166.7 PL=0  +MOVJ EC00398
MACRO1 MJ#(0) ARGF9
ARCON
SMOVL C00399 BC00399 V=10.0  +MOVJ EC00399
SFTON3D P034
SMOVL C00400 BC00400 V=10.0  +MOVJ EC00400
SMOVL C00401 BC00401 V=10.0  +MOVJ EC00401
ARCOF
SMOVL C00402 BC00402 V=800.0  +MOVJ EC00402
SMOVL C00403 BC00403 V=1000.0  +MOVJ EC00403
SMOVL C00404 BC00404 V=1000.0  +MOVJ EC00404
SFTOF3D
'EndPath W4694
MOVJ C00405 BC00405 VJ=100.00  +MOVJ EC00405 VJ=100.00
'Path W4695
SFTOF3D
SFTON3D P032
MOVJ C00406 BC00406 VJ=100.00  +MOVJ EC00406 VJ=100.00
MOVJ C00407 BC00407 VJ=100.00  +MOVJ EC00407 VJ=100.00
SMOVL C00408 BC00408 V=800.0  +MOVJ EC00408
SMOVL C00409 BC00409 V=166.7 PL=0  +MOVJ EC00409
ARCON
SMOVL C00410 BC00410 V=10.5  +MOVJ EC00410
SFTON3D P031
SMOVL C00411 BC00411 V=10.5  +MOVJ EC00411
SMOVL C00412 BC00412 V=10.5  +MOVJ EC00412
ARCOF
SMOVL C00413 BC00413 V=800.0  +MOVJ EC00413
SMOVL C00414 BC00414 V=1000.0  +MOVJ EC00414
SFTOF3D
'EndPath W4695
MOVJ C00415 BC00415 VJ=100.00  +MOVJ EC00415 VJ=100.00
MOVJ C00416 BC00416 VJ=100.00  +MOVJ EC00416 VJ=100.00
'Down
MOVJ C00417 BC00417 VJ=100.00  +MOVJ EC00417 VJ=100.00
'Path W4696
SFTOF3D
SFTON3D P026
MOVJ C00418 BC00418 VJ=100.00  +MOVJ EC00418 VJ=100.00
SMOVL C00419 BC00419 V=800.0  +MOVJ EC00419
SMOVL C00420 BC00420 V=150.0 PL=0  +MOVJ EC00420
MACRO1 MJ#(0) ARGF22
ARCON
SWVON WEV#(108)
SMOVC C00421 BC00421 V=10.0  +MOVJ EC00421
SMOVC C00422 BC00422 V=10.0  +MOVJ EC00422
SMOVC C00423 BC00423 V=10.0  +MOVJ EC00423
SFTON3D P025
SMOVC C00424 BC00424 V=10.0  +MOVJ EC00424
SMOVC C00425 BC00425 V=10.0  +MOVJ EC00425
SMOVC C00426 BC00426 V=10.0  +MOVJ EC00426
SMOVL C00427 BC00427 V=10.0  +MOVJ EC00427
ARCOF
SWVOF
SMOVL C00428 BC00428 V=800.0  +MOVJ EC00428
SMOVL C00429 BC00429 V=1000.0  +MOVJ EC00429
SFTOF3D
'EndPath W4696
MOVJ C00430 BC00430 VJ=100.00  +MOVJ EC00430 VJ=100.00
MOVJ C00431 BC00431 VJ=100.00  +MOVJ EC00431 VJ=100.00
MOVJ C00432 BC00432 VJ=100.00  +MOVJ EC00432 VJ=100.00
MOVJ C00433 BC00433 VJ=100.00  +MOVJ EC00433 VJ=100.00
'Path W4697
SFTOF3D
SFTON3D P022
MOVJ C00434 BC00434 VJ=100.00  +MOVJ EC00434 VJ=100.00
MOVJ C00435 BC00435 VJ=100.00  +MOVJ EC00435 VJ=100.00
SFTON3D P022
SMOVL C00436 BC00436 V=800.0  +MOVJ EC00436
SMOVL C00437 BC00437 V=166.7 PL=0  +MOVJ EC00437
MACRO1 MJ#(0) ARGF9
ARCON
SMOVL C00438 BC00438 V=10.0  +MOVJ EC00438
SMOVL C00439 BC00439 V=10.0  +MOVJ EC00439
SMOVL C00440 BC00440 V=10.0  +MOVJ EC00440
SMOVL C00441 BC00441 V=10.0  +MOVJ EC00441
SMOVL C00442 BC00442 V=10.0  +MOVJ EC00442
SMOVL C00443 BC00443 V=10.0  +MOVJ EC00443
SMOVL C00444 BC00444 V=10.0  +MOVJ EC00444
SMOVL C00445 BC00445 V=10.0  +MOVJ EC00445
SMOVL C00446 BC00446 V=10.0  +MOVJ EC00446
ARCOF
SMOVL C00447 BC00447 V=800.0  +MOVJ EC00447
SMOVL C00448 BC00448 V=1000.0  +MOVJ EC00448
SFTOF3D
'EndPath W4697
'Path W4698
SFTOF3D
SFTON3D P021
SFTOF3D
'EndPath W4698
MOVJ C00449 BC00449 VJ=100.00  +MOVJ EC00449 VJ=100.00
'Path W4699
SFTOF3D
SFTON3D P020
MOVJ C00450 BC00450 VJ=100.00  +MOVJ EC00450 VJ=100.00
SMOVL C00451 BC00451 V=800.0  +MOVJ EC00451
SMOVL C00452 BC00452 V=150.0 PL=0  +MOVJ EC00452
ARCON
SMOVL C00453 BC00453 V=8.3  +MOVJ EC00453
ARCOF
SMOVL C00454 BC00454 V=800.0  +MOVJ EC00454
SFTOF3D
'EndPath W4699
MOVJ C00455 BC00455 VJ=100.00  +MOVJ EC00455 VJ=100.00
MOVJ C00456 BC00456 VJ=100.00  +MOVJ EC00456 VJ=100.00
MOVJ C00457 BC00457 VJ=100.00  +MOVJ EC00457 VJ=100.00
MOVJ C00458 BC00458 VJ=100.00  +MOVJ EC00458 VJ=100.00
'Path W4700
SFTOF3D
SFTON3D P023
MOVJ C00459 BC00459 VJ=100.00  +MOVJ EC00459 VJ=100.00
SMOVL C00460 BC00460 V=800.0  +MOVJ EC00460
'POSPAWANE
SMOVC C00461 BC00461 V=150.0 PL=0  +MOVJ EC00461
MACRO1 MJ#(0) ARGF22
ARCON
SWVON WEV#(108)
SMOVC C00462 BC00462 V=10.0  +MOVJ EC00462
ARCON
SMOVC C00463 BC00463 V=10.0  +MOVJ EC00463
SFTON3D P024
ARCON
SMOVC C00464 BC00464 V=10.0  +MOVJ EC00464
SMOVL C00465 BC00465 V=10.0  +MOVJ EC00465
ARCOF
SWVOF
SMOVL C00466 BC00466 V=800.0  +MOVJ EC00466
SMOVL C00467 BC00467 V=1000.0  +MOVJ EC00467
SFTOF3D
'EndPath W4700
MOVJ C00468 BC00468 VJ=100.00  +MOVJ EC00468 VJ=100.00
MOVJ C00469 BC00469 VJ=100.00  +MOVJ EC00469 VJ=100.00
MOVJ C00470 BC00470 VJ=100.00  +MOVJ EC00470 VJ=100.00
'Path W4701
SFTOF3D
MOVJ C00471 BC00471 VJ=100.00  +MOVJ EC00471 VJ=100.00
MOVL C00472 BC00472 V=666.7  +MOVJ EC00472 VJ=100.00
MOVL C00473 BC00473 V=666.7  +MOVJ EC00473 VJ=100.00
SMOVL C00474 BC00474 V=800.0  +MOVJ EC00474
SFTON3D P046
SMOVL C00475 BC00475 V=150.0 PL=0  +MOVJ EC00475
MACRO1 MJ#(0) ARGF9
ARCON
SFTON3D P047
SMOVL C00476 BC00476 V=10.0  +MOVJ EC00476
SMOVC C00477 BC00477 V=13.3  +MOVJ EC00477
SMOVC C00478 BC00478 V=13.3  +MOVJ EC00478
SMOVC C00479 BC00479 V=13.3  +MOVJ EC00479
SFTON3D P046
SMOVL C00480 BC00480 V=10.0  +MOVJ EC00480
SMOVC C00481 BC00481 V=13.3  +MOVJ EC00481
SMOVC C00482 BC00482 V=13.3  +MOVJ EC00482
SMOVC C00483 BC00483 V=13.3  +MOVJ EC00483
ARCOF
SMOVL C00484 BC00484 V=166.7  +MOVJ EC00484
SFTOF3D
MOVL C00485 BC00485 V=666.7  +MOVJ EC00485 VJ=100.00
MOVL C00486 BC00486 V=666.7  +MOVJ EC00486 VJ=100.00
SMOVL C00487 BC00487 V=800.0  +MOVJ EC00487
SFTON3D P044
SMOVL C00488 BC00488 V=150.0 PL=0  +MOVJ EC00488
MACRO1 MJ#(0) ARGF9
ARCON
SFTON3D P045
SMOVL C00489 BC00489 V=10.0  +MOVJ EC00489
SMOVC C00490 BC00490 V=13.3  +MOVJ EC00490
SMOVC C00491 BC00491 V=13.3  +MOVJ EC00491
SMOVC C00492 BC00492 V=13.3  +MOVJ EC00492
SFTON3D P044
SMOVL C00493 BC00493 V=10.0  +MOVJ EC00493
SMOVL C00494 BC00494 V=10.0  +MOVJ EC00494
SMOVC C00495 BC00495 V=13.3  +MOVJ EC00495
SMOVC C00496 BC00496 V=13.3  +MOVJ EC00496
SMOVC C00497 BC00497 V=13.3  +MOVJ EC00497
ARCOF
SMOVL C00498 BC00498 V=166.7  +MOVJ EC00498
SFTOF3D
SMOVL C00499 BC00499 V=666.7  +MOVJ EC00499
MOVJ C00500 BC00500 VJ=100.00  +MOVJ EC00500 VJ=100.00
MOVJ C00501 BC00501 VJ=100.00  +MOVJ EC00501 VJ=100.00
SMOVL C00502 BC00502 V=800.0  +MOVJ EC00502
SFTON3D P048
SMOVL C00503 BC00503 V=150.0 PL=0  +MOVJ EC00503
MACRO1 MJ#(0) ARGF9
ARCON
SFTON3D P049
SMOVL C00504 BC00504 V=10.0  +MOVJ EC00504
SMOVC C00505 BC00505 V=13.3  +MOVJ EC00505
SMOVC C00506 BC00506 V=13.3  +MOVJ EC00506
SMOVC C00507 BC00507 V=13.3  +MOVJ EC00507
SFTON3D P048
SMOVL C00508 BC00508 V=10.0  +MOVJ EC00508
SMOVL C00509 BC00509 V=10.0  +MOVJ EC00509
SMOVC C00510 BC00510 V=13.3  +MOVJ EC00510
SMOVC C00511 BC00511 V=13.3  +MOVJ EC00511
SMOVC C00512 BC00512 V=13.3  +MOVJ EC00512
ARCOF
SMOVL C00513 BC00513 V=166.7  +MOVJ EC00513
SFTOF3D
MOVJ C00514 BC00514 VJ=50.00  +MOVJ EC00514 VJ=0.78
SFTON3D P057
SMOVL C00515 BC00515 V=150.0 PL=0  +MOVJ EC00515
MACRO1 MJ#(0) ARGF9
ARCON
SFTON3D P058
SMOVL C00516 BC00516 V=10.0  +MOVJ EC00516
SMOVC C00517 BC00517 V=13.3  +MOVJ EC00517
SMOVC C00518 BC00518 V=13.3  +MOVJ EC00518
SMOVC C00519 BC00519 V=13.3  +MOVJ EC00519
SFTON3D P057
SMOVL C00520 BC00520 V=10.0  +MOVJ EC00520
SMOVL C00521 BC00521 V=10.0  +MOVJ EC00521
SMOVC C00522 BC00522 V=13.3  +MOVJ EC00522
SMOVC C00523 BC00523 V=13.3  +MOVJ EC00523
SMOVC C00524 BC00524 V=13.3  +MOVJ EC00524
ARCOF
SMOVL C00525 BC00525 V=166.7  +MOVJ EC00525
SFTOF3D
MOVJ C00526 BC00526 VJ=30.00  +MOVJ EC00526 VJ=50.00
SFTON3D P053
SMOVL C00527 BC00527 V=166.7  +MOVJ EC00527
SMOVL C00528 BC00528 V=150.0 PL=0  +MOVJ EC00528
MACRO1 MJ#(0) ARGF9
ARCON
SFTON3D P054
SMOVL C00529 BC00529 V=10.0  +MOVJ EC00529
SMOVC C00530 BC00530 V=13.3  +MOVJ EC00530
SMOVC C00531 BC00531 V=13.3  +MOVJ EC00531
SMOVC C00532 BC00532 V=13.3  +MOVJ EC00532
SFTON3D P053
SMOVL C00533 BC00533 V=10.0  +MOVJ EC00533
SMOVL C00534 BC00534 V=10.0  +MOVJ EC00534
SMOVC C00535 BC00535 V=13.3  +MOVJ EC00535
SMOVC C00536 BC00536 V=13.3  +MOVJ EC00536
SMOVC C00537 BC00537 V=13.3  +MOVJ EC00537
ARCOF
SMOVL C00538 BC00538 V=166.7  +MOVJ EC00538
SFTOF3D
SMOVL C00539 BC00539 V=666.7  +MOVJ EC00539
SFTON3D P056
SMOVL C00540 BC00540 V=150.0 PL=0  +MOVJ EC00540
MACRO1 MJ#(0) ARGF9
ARCON
SFTON3D P055
SMOVL C00541 BC00541 V=10.0  +MOVJ EC00541
SMOVC C00542 BC00542 V=13.3  +MOVJ EC00542
SMOVC C00543 BC00543 V=13.3  +MOVJ EC00543
SMOVC C00544 BC00544 V=13.3  +MOVJ EC00544
SFTON3D P056
SMOVL C00545 BC00545 V=10.0  +MOVJ EC00545
SMOVL C00546 BC00546 V=10.0  +MOVJ EC00546
SMOVC C00547 BC00547 V=13.3  +MOVJ EC00547
SMOVC C00548 BC00548 V=13.3  +MOVJ EC00548
SMOVC C00549 BC00549 V=13.3  +MOVJ EC00549
ARCOF
SMOVL C00550 BC00550 V=166.7  +MOVJ EC00550
SFTOF3D
MOVL C00551 BC00551 V=666.7  +MOVJ EC00551 VJ=30.00
SFTON3D P052
SMOVL C00552 BC00552 V=150.0 PL=0  +MOVJ EC00552
ARCON
SMOVL C00553 BC00553 V=10.0  +MOVJ EC00553
SMOVC C00554 BC00554 V=13.3  +MOVJ EC00554
SFTON3D P051
SMOVC C00555 BC00555 V=13.3  +MOVJ EC00555
SMOVC C00556 BC00556 V=13.3  +MOVJ EC00556
SFTON3D P050
SMOVL C00557 BC00557 V=10.0  +MOVJ EC00557
ARCOF
SMOVL C00558 BC00558 V=166.7  +MOVJ EC00558
SFTOF3D
SMOVL C00559 BC00559 V=1000.0  +MOVJ EC00559
SMOVL C00560 BC00560 V=1000.0  +MOVJ EC00560
SFTON3D P041
SMOVL C00561 BC00561 V=100.0  +MOVJ EC00561
SMOVL C00562 BC00562 V=1000.0  +MOVJ EC00562
SMOVL C00563 BC00563 V=150.0 PL=0  +MOVJ EC00563
ARCON
SMOVL C00564 BC00564 V=10.0  +MOVJ EC00564
SMOVC C00565 BC00565 V=13.3  +MOVJ EC00565
SMOVC C00566 BC00566 V=13.3  +MOVJ EC00566
SMOVC C00567 BC00567 V=13.3  +MOVJ EC00567
SFTON3D P042
SMOVL C00568 BC00568 V=10.0  +MOVJ EC00568
SFTON3D P043
SMOVL C00569 BC00569 V=10.0  +MOVJ EC00569
SMOVC C00570 BC00570 V=13.3  +MOVJ EC00570
SMOVC C00571 BC00571 V=13.3  +MOVJ EC00571
SMOVC C00572 BC00572 V=13.3  +MOVJ EC00572
ARCOF
SMOVL C00573 BC00573 V=166.7  +MOVJ EC00573
SFTOF3D
SMOVL C00574 BC00574 V=1000.0  +MOVJ EC00574
END
